ABB RAPID module: robotPath.mod

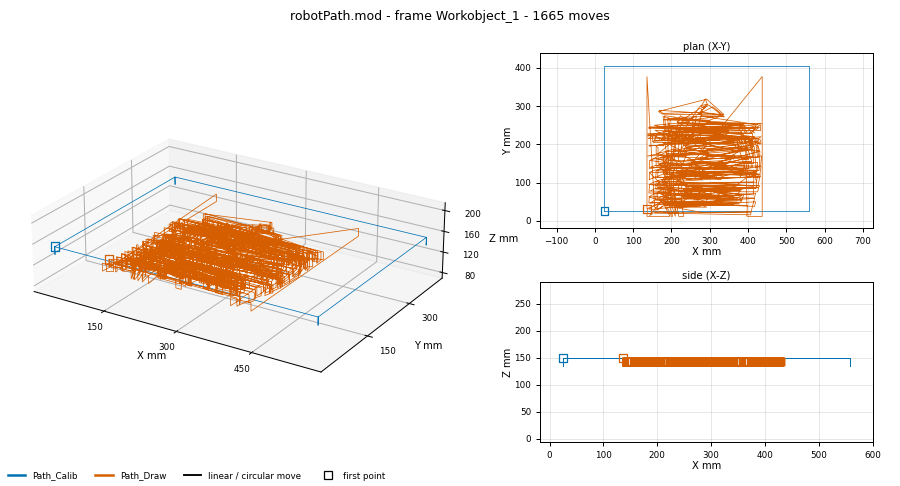
[picture p0: tool path of robotPath.mod in frame Workobject_1, 1665 of 1667 moves have a stored position in this frame; points joined in program order, loops and branches not executed]
MODULE MainModule
    CONST jointtarget home:=[[-90,40,10,0,40,90],[9E+09,9E+09,9E+09,9E+09,9E+09,9E+09]];
    CONST robtarget calib_1:=[[25,25,149.5],[0,0,1,0],[0,0,0,0],[9E+09,9E+09,9E+09,9E+09,9E+09,9E+09]];
    CONST robtarget calib_1d:=[[25,25,134.5],[0,0,1,0],[0,0,0,0],[9E+09,9E+09,9E+09,9E+09,9E+09,9E+09]];
    CONST robtarget calib_2:=[[558,25,149.5],[0,0,1,0],[0,0,0,0],[9E+09,9E+09,9E+09,9E+09,9E+09,9E+09]];
    CONST robtarget calib_2d:=[[558,25,134.5],[0,0,1,0],[0,0,0,0],[9E+09,9E+09,9E+09,9E+09,9E+09,9E+09]];
    CONST robtarget calib_3:=[[558,406,149.5],[0,0,1,0],[0,0,0,0],[9E+09,9E+09,9E+09,9E+09,9E+09,9E+09]];
    CONST robtarget calib_3d:=[[558,406,134.5],[0,0,1,0],[0,0,0,0],[9E+09,9E+09,9E+09,9E+09,9E+09,9E+09]];
    CONST robtarget calib_4:=[[25,406,149.5],[0,0,1,0],[0,0,0,0],[9E+09,9E+09,9E+09,9E+09,9E+09,9E+09]];
    CONST robtarget calib_4d:=[[25,406,134.5],[0,0,1,0],[0,0,0,0],[9E+09,9E+09,9E+09,9E+09,9E+09,9E+09]];
    CONST robtarget point_0_clearance:=[[137,31,149.5],[0,0,1,0],[0, 0, 0, 0],[9E+09,9E+09,9E+09,9E+09,9E+09,9E+09]];
    CONST robtarget point_0_contact:=[[137,31,134.5],[0,0,1,0],[0, 0, 0, 0],[9E+09,9E+09,9E+09,9E+09,9E+09,9E+09]];
    CONST robtarget point_1_contact:=[[136,12,134.5],[0,0,1,0],[0, 0, 0, 0],[9E+09,9E+09,9E+09,9E+09,9E+09,9E+09]];
    CONST robtarget point_1_clearance:=[[136,12,149.5],[0,0,1,0],[0, 0, 0, 0],[9E+09,9E+09,9E+09,9E+09,9E+09,9E+09]];
    CONST robtarget point_2_clearance:=[[196,12,149.5],[0,0,1,0],[0, 0, 0, 0],[9E+09,9E+09,9E+09,9E+09,9E+09,9E+09]];
    CONST robtarget point_2_contact:=[[196,12,134.5],[0,0,1,0],[0, 0, 0, 0],[9E+09,9E+09,9E+09,9E+09,9E+09,9E+09]];
    CONST robtarget point_3_contact:=[[185,34,134.5],[0,0,1,0],[0, 0, 0, 0],[9E+09,9E+09,9E+09,9E+09,9E+09,9E+09]];
    CONST robtarget point_3_clearance:=[[185,34,149.5],[0,0,1,0],[0, 0, 0, 0],[9E+09,9E+09,9E+09,9E+09,9E+09,9E+09]];
    CONST robtarget point_4_clearance:=[[192,30,149.5],[0,0,1,0],[0, 0, 0, 0],[9E+09,9E+09,9E+09,9E+09,9E+09,9E+09]];
    CONST robtarget point_4_contact:=[[192,30,134.5],[0,0,1,0],[0, 0, 0, 0],[9E+09,9E+09,9E+09,9E+09,9E+09,9E+09]];
    CONST robtarget point_5_contact:=[[200,12,134.5],[0,0,1,0],[0, 0, 0, 0],[9E+09,9E+09,9E+09,9E+09,9E+09,9E+09]];
    CONST robtarget point_5_clearance:=[[200,12,149.5],[0,0,1,0],[0, 0, 0, 0],[9E+09,9E+09,9E+09,9E+09,9E+09,9E+09]];
    CONST robtarget point_6_clearance:=[[203,12,149.5],[0,0,1,0],[0, 0, 0, 0],[9E+09,9E+09,9E+09,9E+09,9E+09,9E+09]];
    CONST robtarget point_6_contact:=[[203,12,134.5],[0,0,1,0],[0, 0, 0, 0],[9E+09,9E+09,9E+09,9E+09,9E+09,9E+09]];
    CONST robtarget point_7_contact:=[[195,41,134.5],[0,0,1,0],[0, 0, 0, 0],[9E+09,9E+09,9E+09,9E+09,9E+09,9E+09]];
    CONST robtarget point_7_clearance:=[[195,41,149.5],[0,0,1,0],[0, 0, 0, 0],[9E+09,9E+09,9E+09,9E+09,9E+09,9E+09]];
    CONST robtarget point_8_clearance:=[[197,51,149.5],[0,0,1,0],[0, 0, 0, 0],[9E+09,9E+09,9E+09,9E+09,9E+09,9E+09]];
    CONST robtarget point_8_contact:=[[197,51,134.5],[0,0,1,0],[0, 0, 0, 0],[9E+09,9E+09,9E+09,9E+09,9E+09,9E+09]];
    CONST robtarget point_9_contact:=[[210,12,134.5],[0,0,1,0],[0, 0, 0, 0],[9E+09,9E+09,9E+09,9E+09,9E+09,9E+09]];
    CONST robtarget point_9_clearance:=[[210,12,149.5],[0,0,1,0],[0, 0, 0, 0],[9E+09,9E+09,9E+09,9E+09,9E+09,9E+09]];
    CONST robtarget point_10_clearance:=[[206,86,149.5],[0,0,1,0],[0, 0, 0, 0],[9E+09,9E+09,9E+09,9E+09,9E+09,9E+09]];
    CONST robtarget point_10_contact:=[[206,86,134.5],[0,0,1,0],[0, 0, 0, 0],[9E+09,9E+09,9E+09,9E+09,9E+09,9E+09]];
    CONST robtarget point_11_contact:=[[219,12,134.5],[0,0,1,0],[0, 0, 0, 0],[9E+09,9E+09,9E+09,9E+09,9E+09,9E+09]];
    CONST robtarget point_11_clearance:=[[219,12,149.5],[0,0,1,0],[0, 0, 0, 0],[9E+09,9E+09,9E+09,9E+09,9E+09,9E+09]];
    CONST robtarget point_12_clearance:=[[232,12,149.5],[0,0,1,0],[0, 0, 0, 0],[9E+09,9E+09,9E+09,9E+09,9E+09,9E+09]];
    CONST robtarget point_12_contact:=[[232,12,134.5],[0,0,1,0],[0, 0, 0, 0],[9E+09,9E+09,9E+09,9E+09,9E+09,9E+09]];
    CONST robtarget point_13_contact:=[[226,51,134.5],[0,0,1,0],[0, 0, 0, 0],[9E+09,9E+09,9E+09,9E+09,9E+09,9E+09]];
    CONST robtarget point_13_clearance:=[[226,51,149.5],[0,0,1,0],[0, 0, 0, 0],[9E+09,9E+09,9E+09,9E+09,9E+09,9E+09]];
    CONST robtarget point_14_clearance:=[[398,40,149.5],[0,0,1,0],[0, 0, 0, 0],[9E+09,9E+09,9E+09,9E+09,9E+09,9E+09]];
    CONST robtarget point_14_contact:=[[398,40,134.5],[0,0,1,0],[0, 0, 0, 0],[9E+09,9E+09,9E+09,9E+09,9E+09,9E+09]];
    CONST robtarget point_15_contact:=[[397,12,134.5],[0,0,1,0],[0, 0, 0, 0],[9E+09,9E+09,9E+09,9E+09,9E+09,9E+09]];
    CONST robtarget point_15_clearance:=[[397,12,149.5],[0,0,1,0],[0, 0, 0, 0],[9E+09,9E+09,9E+09,9E+09,9E+09,9E+09]];
    CONST robtarget point_16_clearance:=[[437,12,149.5],[0,0,1,0],[0, 0, 0, 0],[9E+09,9E+09,9E+09,9E+09,9E+09,9E+09]];
    CONST robtarget point_16_contact:=[[437,12,134.5],[0,0,1,0],[0, 0, 0, 0],[9E+09,9E+09,9E+09,9E+09,9E+09,9E+09]];
    CONST robtarget point_17_contact:=[[437,377,134.5],[0,0,1,0],[0, 0, 0, 0],[9E+09,9E+09,9E+09,9E+09,9E+09,9E+09]];
    CONST robtarget point_17_clearance:=[[437,377,149.5],[0,0,1,0],[0, 0, 0, 0],[9E+09,9E+09,9E+09,9E+09,9E+09,9E+09]];
    CONST robtarget point_18_clearance:=[[143,14,149.5],[0,0,1,0],[0, 0, 0, 0],[9E+09,9E+09,9E+09,9E+09,9E+09,9E+09]];
    CONST robtarget point_18_contact:=[[143,14,134.5],[0,0,1,0],[0, 0, 0, 0],[9E+09,9E+09,9E+09,9E+09,9E+09,9E+09]];
    CONST robtarget point_19_contact:=[[153,21,134.5],[0,0,1,0],[0, 0, 0, 0],[9E+09,9E+09,9E+09,9E+09,9E+09,9E+09]];
    CONST robtarget point_19_clearance:=[[153,21,149.5],[0,0,1,0],[0, 0, 0, 0],[9E+09,9E+09,9E+09,9E+09,9E+09,9E+09]];
    CONST robtarget point_20_clearance:=[[407,16,149.5],[0,0,1,0],[0, 0, 0, 0],[9E+09,9E+09,9E+09,9E+09,9E+09,9E+09]];
    CONST robtarget point_20_contact:=[[407,16,134.5],[0,0,1,0],[0, 0, 0, 0],[9E+09,9E+09,9E+09,9E+09,9E+09,9E+09]];
    CONST robtarget point_21_contact:=[[408,23,134.5],[0,0,1,0],[0, 0, 0, 0],[9E+09,9E+09,9E+09,9E+09,9E+09,9E+09]];
    CONST robtarget point_21_clearance:=[[408,23,149.5],[0,0,1,0],[0, 0, 0, 0],[9E+09,9E+09,9E+09,9E+09,9E+09,9E+09]];
    CONST robtarget point_22_clearance:=[[157,21,149.5],[0,0,1,0],[0, 0, 0, 0],[9E+09,9E+09,9E+09,9E+09,9E+09,9E+09]];
    CONST robtarget point_22_contact:=[[157,21,134.5],[0,0,1,0],[0, 0, 0, 0],[9E+09,9E+09,9E+09,9E+09,9E+09,9E+09]];
    CONST robtarget point_23_contact:=[[157,26,134.5],[0,0,1,0],[0, 0, 0, 0],[9E+09,9E+09,9E+09,9E+09,9E+09,9E+09]];
    CONST robtarget point_23_clearance:=[[157,26,149.5],[0,0,1,0],[0, 0, 0, 0],[9E+09,9E+09,9E+09,9E+09,9E+09,9E+09]];
    CONST robtarget point_24_clearance:=[[213,21,149.5],[0,0,1,0],[0, 0, 0, 0],[9E+09,9E+09,9E+09,9E+09,9E+09,9E+09]];
    CONST robtarget point_24_contact:=[[213,21,134.5],[0,0,1,0],[0, 0, 0, 0],[9E+09,9E+09,9E+09,9E+09,9E+09,9E+09]];
    CONST robtarget point_25_contact:=[[210,35,134.5],[0,0,1,0],[0, 0, 0, 0],[9E+09,9E+09,9E+09,9E+09,9E+09,9E+09]];
    CONST robtarget point_25_clearance:=[[210,35,149.5],[0,0,1,0],[0, 0, 0, 0],[9E+09,9E+09,9E+09,9E+09,9E+09,9E+09]];
    CONST robtarget point_26_clearance:=[[281,22,149.5],[0,0,1,0],[0, 0, 0, 0],[9E+09,9E+09,9E+09,9E+09,9E+09,9E+09]];
    CONST robtarget point_26_contact:=[[281,22,134.5],[0,0,1,0],[0, 0, 0, 0],[9E+09,9E+09,9E+09,9E+09,9E+09,9E+09]];
    CONST robtarget point_27_contact:=[[292,22,134.5],[0,0,1,0],[0, 0, 0, 0],[9E+09,9E+09,9E+09,9E+09,9E+09,9E+09]];
    CONST robtarget point_27_clearance:=[[292,22,149.5],[0,0,1,0],[0, 0, 0, 0],[9E+09,9E+09,9E+09,9E+09,9E+09,9E+09]];
    CONST robtarget point_28_clearance:=[[408,24,149.5],[0,0,1,0],[0, 0, 0, 0],[9E+09,9E+09,9E+09,9E+09,9E+09,9E+09]];
    CONST robtarget point_28_contact:=[[408,24,134.5],[0,0,1,0],[0, 0, 0, 0],[9E+09,9E+09,9E+09,9E+09,9E+09,9E+09]];
    CONST robtarget point_29_contact:=[[417,59,134.5],[0,0,1,0],[0, 0, 0, 0],[9E+09,9E+09,9E+09,9E+09,9E+09,9E+09]];
    CONST robtarget point_29_clearance:=[[417,59,149.5],[0,0,1,0],[0, 0, 0, 0],[9E+09,9E+09,9E+09,9E+09,9E+09,9E+09]];
    CONST robtarget point_30_clearance:=[[156,42,149.5],[0,0,1,0],[0, 0, 0, 0],[9E+09,9E+09,9E+09,9E+09,9E+09,9E+09]];
    CONST robtarget point_30_contact:=[[156,42,134.5],[0,0,1,0],[0, 0, 0, 0],[9E+09,9E+09,9E+09,9E+09,9E+09,9E+09]];
    CONST robtarget point_31_contact:=[[141,31,134.5],[0,0,1,0],[0, 0, 0, 0],[9E+09,9E+09,9E+09,9E+09,9E+09,9E+09]];
    CONST robtarget point_31_clearance:=[[141,31,149.5],[0,0,1,0],[0, 0, 0, 0],[9E+09,9E+09,9E+09,9E+09,9E+09,9E+09]];
    CONST robtarget point_32_clearance:=[[166,30,149.5],[0,0,1,0],[0, 0, 0, 0],[9E+09,9E+09,9E+09,9E+09,9E+09,9E+09]];
    CONST robtarget point_32_contact:=[[166,30,134.5],[0,0,1,0],[0, 0, 0, 0],[9E+09,9E+09,9E+09,9E+09,9E+09,9E+09]];
    CONST robtarget point_33_contact:=[[178,39,134.5],[0,0,1,0],[0, 0, 0, 0],[9E+09,9E+09,9E+09,9E+09,9E+09,9E+09]];
    CONST robtarget point_33_clearance:=[[178,39,149.5],[0,0,1,0],[0, 0, 0, 0],[9E+09,9E+09,9E+09,9E+09,9E+09,9E+09]];
    CONST robtarget point_34_clearance:=[[164,31,149.5],[0,0,1,0],[0, 0, 0, 0],[9E+09,9E+09,9E+09,9E+09,9E+09,9E+09]];
    CONST robtarget point_34_contact:=[[164,31,134.5],[0,0,1,0],[0, 0, 0, 0],[9E+09,9E+09,9E+09,9E+09,9E+09,9E+09]];
    CONST robtarget point_35_contact:=[[156,36,134.5],[0,0,1,0],[0, 0, 0, 0],[9E+09,9E+09,9E+09,9E+09,9E+09,9E+09]];
    CONST robtarget point_35_clearance:=[[156,36,149.5],[0,0,1,0],[0, 0, 0, 0],[9E+09,9E+09,9E+09,9E+09,9E+09,9E+09]];
    CONST robtarget point_36_clearance:=[[136,377,149.5],[0,0,1,0],[0, 0, 0, 0],[9E+09,9E+09,9E+09,9E+09,9E+09,9E+09]];
    CONST robtarget point_36_contact:=[[136,377,134.5],[0,0,1,0],[0, 0, 0, 0],[9E+09,9E+09,9E+09,9E+09,9E+09,9E+09]];
    CONST robtarget point_37_contact:=[[136,32,134.5],[0,0,1,0],[0, 0, 0, 0],[9E+09,9E+09,9E+09,9E+09,9E+09,9E+09]];
    CONST robtarget point_37_clearance:=[[136,32,149.5],[0,0,1,0],[0, 0, 0, 0],[9E+09,9E+09,9E+09,9E+09,9E+09,9E+09]];
    CONST robtarget point_38_clearance:=[[164,43,149.5],[0,0,1,0],[0, 0, 0, 0],[9E+09,9E+09,9E+09,9E+09,9E+09,9E+09]];
    CONST robtarget point_38_contact:=[[164,43,134.5],[0,0,1,0],[0, 0, 0, 0],[9E+09,9E+09,9E+09,9E+09,9E+09,9E+09]];
    CONST robtarget point_39_contact:=[[164,32,134.5],[0,0,1,0],[0, 0, 0, 0],[9E+09,9E+09,9E+09,9E+09,9E+09,9E+09]];
    CONST robtarget point_39_clearance:=[[164,32,149.5],[0,0,1,0],[0, 0, 0, 0],[9E+09,9E+09,9E+09,9E+09,9E+09,9E+09]];
    CONST robtarget point_40_clearance:=[[241,40,149.5],[0,0,1,0],[0, 0, 0, 0],[9E+09,9E+09,9E+09,9E+09,9E+09,9E+09]];
    CONST robtarget point_40_contact:=[[241,40,134.5],[0,0,1,0],[0, 0, 0, 0],[9E+09,9E+09,9E+09,9E+09,9E+09,9E+09]];
    CONST robtarget point_41_contact:=[[278,39,134.5],[0,0,1,0],[0, 0, 0, 0],[9E+09,9E+09,9E+09,9E+09,9E+09,9E+09]];
    CONST robtarget point_41_clearance:=[[278,39,149.5],[0,0,1,0],[0, 0, 0, 0],[9E+09,9E+09,9E+09,9E+09,9E+09,9E+09]];
    CONST robtarget point_42_clearance:=[[185,34,149.5],[0,0,1,0],[0, 0, 0, 0],[9E+09,9E+09,9E+09,9E+09,9E+09,9E+09]];
    CONST robtarget point_42_contact:=[[185,34,134.5],[0,0,1,0],[0, 0, 0, 0],[9E+09,9E+09,9E+09,9E+09,9E+09,9E+09]];
    CONST robtarget point_43_contact:=[[180,43,134.5],[0,0,1,0],[0, 0, 0, 0],[9E+09,9E+09,9E+09,9E+09,9E+09,9E+09]];
    CONST robtarget point_43_clearance:=[[180,43,149.5],[0,0,1,0],[0, 0, 0, 0],[9E+09,9E+09,9E+09,9E+09,9E+09,9E+09]];
    CONST robtarget point_44_clearance:=[[276,42,149.5],[0,0,1,0],[0, 0, 0, 0],[9E+09,9E+09,9E+09,9E+09,9E+09,9E+09]];
    CONST robtarget point_44_contact:=[[276,42,134.5],[0,0,1,0],[0, 0, 0, 0],[9E+09,9E+09,9E+09,9E+09,9E+09,9E+09]];
    CONST robtarget point_45_contact:=[[292,36,134.5],[0,0,1,0],[0, 0, 0, 0],[9E+09,9E+09,9E+09,9E+09,9E+09,9E+09]];
    CONST robtarget point_45_clearance:=[[292,36,149.5],[0,0,1,0],[0, 0, 0, 0],[9E+09,9E+09,9E+09,9E+09,9E+09,9E+09]];
    CONST robtarget point_46_clearance:=[[196,36,149.5],[0,0,1,0],[0, 0, 0, 0],[9E+09,9E+09,9E+09,9E+09,9E+09,9E+09]];
    CONST robtarget point_46_contact:=[[196,36,134.5],[0,0,1,0],[0, 0, 0, 0],[9E+09,9E+09,9E+09,9E+09,9E+09,9E+09]];
    CONST robtarget point_47_contact:=[[192,42,134.5],[0,0,1,0],[0, 0, 0, 0],[9E+09,9E+09,9E+09,9E+09,9E+09,9E+09]];
    CONST robtarget point_47_clearance:=[[192,42,149.5],[0,0,1,0],[0, 0, 0, 0],[9E+09,9E+09,9E+09,9E+09,9E+09,9E+09]];
    CONST robtarget point_48_clearance:=[[231,41,149.5],[0,0,1,0],[0, 0, 0, 0],[9E+09,9E+09,9E+09,9E+09,9E+09,9E+09]];
    CONST robtarget point_48_contact:=[[231,41,134.5],[0,0,1,0],[0, 0, 0, 0],[9E+09,9E+09,9E+09,9E+09,9E+09,9E+09]];
    CONST robtarget point_49_contact:=[[236,38,134.5],[0,0,1,0],[0, 0, 0, 0],[9E+09,9E+09,9E+09,9E+09,9E+09,9E+09]];
    CONST robtarget point_49_clearance:=[[236,38,149.5],[0,0,1,0],[0, 0, 0, 0],[9E+09,9E+09,9E+09,9E+09,9E+09,9E+09]];
    CONST robtarget point_50_clearance:=[[239,37,149.5],[0,0,1,0],[0, 0, 0, 0],[9E+09,9E+09,9E+09,9E+09,9E+09,9E+09]];
    CONST robtarget point_50_contact:=[[239,37,134.5],[0,0,1,0],[0, 0, 0, 0],[9E+09,9E+09,9E+09,9E+09,9E+09,9E+09]];
    CONST robtarget point_51_contact:=[[234,45,134.5],[0,0,1,0],[0, 0, 0, 0],[9E+09,9E+09,9E+09,9E+09,9E+09,9E+09]];
    CONST robtarget point_51_clearance:=[[234,45,149.5],[0,0,1,0],[0, 0, 0, 0],[9E+09,9E+09,9E+09,9E+09,9E+09,9E+09]];
    CONST robtarget point_52_clearance:=[[348,42,149.5],[0,0,1,0],[0, 0, 0, 0],[9E+09,9E+09,9E+09,9E+09,9E+09,9E+09]];
    CONST robtarget point_52_contact:=[[348,42,134.5],[0,0,1,0],[0, 0, 0, 0],[9E+09,9E+09,9E+09,9E+09,9E+09,9E+09]];
    CONST robtarget point_53_contact:=[[362,42,134.5],[0,0,1,0],[0, 0, 0, 0],[9E+09,9E+09,9E+09,9E+09,9E+09,9E+09]];
    CONST robtarget point_53_clearance:=[[362,42,149.5],[0,0,1,0],[0, 0, 0, 0],[9E+09,9E+09,9E+09,9E+09,9E+09,9E+09]];
    CONST robtarget point_54_clearance:=[[239,39,149.5],[0,0,1,0],[0, 0, 0, 0],[9E+09,9E+09,9E+09,9E+09,9E+09,9E+09]];
    CONST robtarget point_54_contact:=[[239,39,134.5],[0,0,1,0],[0, 0, 0, 0],[9E+09,9E+09,9E+09,9E+09,9E+09,9E+09]];
    CONST robtarget point_55_contact:=[[244,44,134.5],[0,0,1,0],[0, 0, 0, 0],[9E+09,9E+09,9E+09,9E+09,9E+09,9E+09]];
    CONST robtarget point_55_clearance:=[[244,44,149.5],[0,0,1,0],[0, 0, 0, 0],[9E+09,9E+09,9E+09,9E+09,9E+09,9E+09]];
    CONST robtarget point_56_clearance:=[[330,44,149.5],[0,0,1,0],[0, 0, 0, 0],[9E+09,9E+09,9E+09,9E+09,9E+09,9E+09]];
    CONST robtarget point_56_contact:=[[330,44,134.5],[0,0,1,0],[0, 0, 0, 0],[9E+09,9E+09,9E+09,9E+09,9E+09,9E+09]];
    CONST robtarget point_57_contact:=[[349,46,134.5],[0,0,1,0],[0, 0, 0, 0],[9E+09,9E+09,9E+09,9E+09,9E+09,9E+09]];
    CONST robtarget point_57_clearance:=[[349,46,149.5],[0,0,1,0],[0, 0, 0, 0],[9E+09,9E+09,9E+09,9E+09,9E+09,9E+09]];
    CONST robtarget point_58_clearance:=[[420,50,149.5],[0,0,1,0],[0, 0, 0, 0],[9E+09,9E+09,9E+09,9E+09,9E+09,9E+09]];
    CONST robtarget point_58_contact:=[[420,50,134.5],[0,0,1,0],[0, 0, 0, 0],[9E+09,9E+09,9E+09,9E+09,9E+09,9E+09]];
    CONST robtarget point_59_contact:=[[417,38,134.5],[0,0,1,0],[0, 0, 0, 0],[9E+09,9E+09,9E+09,9E+09,9E+09,9E+09]];
    CONST robtarget point_59_clearance:=[[417,38,149.5],[0,0,1,0],[0, 0, 0, 0],[9E+09,9E+09,9E+09,9E+09,9E+09,9E+09]];
    CONST robtarget point_60_clearance:=[[182,48,149.5],[0,0,1,0],[0, 0, 0, 0],[9E+09,9E+09,9E+09,9E+09,9E+09,9E+09]];
    CONST robtarget point_60_contact:=[[182,48,134.5],[0,0,1,0],[0, 0, 0, 0],[9E+09,9E+09,9E+09,9E+09,9E+09,9E+09]];
    CONST robtarget point_61_contact:=[[185,39,134.5],[0,0,1,0],[0, 0, 0, 0],[9E+09,9E+09,9E+09,9E+09,9E+09,9E+09]];
    CONST robtarget point_61_clearance:=[[185,39,149.5],[0,0,1,0],[0, 0, 0, 0],[9E+09,9E+09,9E+09,9E+09,9E+09,9E+09]];
    CONST robtarget point_62_clearance:=[[287,44,149.5],[0,0,1,0],[0, 0, 0, 0],[9E+09,9E+09,9E+09,9E+09,9E+09,9E+09]];
    CONST robtarget point_62_contact:=[[287,44,134.5],[0,0,1,0],[0, 0, 0, 0],[9E+09,9E+09,9E+09,9E+09,9E+09,9E+09]];
    CONST robtarget point_63_contact:=[[295,41,134.5],[0,0,1,0],[0, 0, 0, 0],[9E+09,9E+09,9E+09,9E+09,9E+09,9E+09]];
    CONST robtarget point_63_clearance:=[[295,41,149.5],[0,0,1,0],[0, 0, 0, 0],[9E+09,9E+09,9E+09,9E+09,9E+09,9E+09]];
    CONST robtarget point_64_clearance:=[[293,41,149.5],[0,0,1,0],[0, 0, 0, 0],[9E+09,9E+09,9E+09,9E+09,9E+09,9E+09]];
    CONST robtarget point_64_contact:=[[293,41,134.5],[0,0,1,0],[0, 0, 0, 0],[9E+09,9E+09,9E+09,9E+09,9E+09,9E+09]];
    CONST robtarget point_65_contact:=[[300,42,134.5],[0,0,1,0],[0, 0, 0, 0],[9E+09,9E+09,9E+09,9E+09,9E+09,9E+09]];
    CONST robtarget point_65_clearance:=[[300,42,149.5],[0,0,1,0],[0, 0, 0, 0],[9E+09,9E+09,9E+09,9E+09,9E+09,9E+09]];
    CONST robtarget point_66_clearance:=[[396,113,149.5],[0,0,1,0],[0, 0, 0, 0],[9E+09,9E+09,9E+09,9E+09,9E+09,9E+09]];
    CONST robtarget point_66_contact:=[[396,113,134.5],[0,0,1,0],[0, 0, 0, 0],[9E+09,9E+09,9E+09,9E+09,9E+09,9E+09]];
    CONST robtarget point_67_contact:=[[397,40,134.5],[0,0,1,0],[0, 0, 0, 0],[9E+09,9E+09,9E+09,9E+09,9E+09,9E+09]];
    CONST robtarget point_67_clearance:=[[397,40,149.5],[0,0,1,0],[0, 0, 0, 0],[9E+09,9E+09,9E+09,9E+09,9E+09,9E+09]];
    CONST robtarget point_68_clearance:=[[179,41,149.5],[0,0,1,0],[0, 0, 0, 0],[9E+09,9E+09,9E+09,9E+09,9E+09,9E+09]];
    CONST robtarget point_68_contact:=[[179,41,134.5],[0,0,1,0],[0, 0, 0, 0],[9E+09,9E+09,9E+09,9E+09,9E+09,9E+09]];
    CONST robtarget point_69_contact:=[[178,51,134.5],[0,0,1,0],[0, 0, 0, 0],[9E+09,9E+09,9E+09,9E+09,9E+09,9E+09]];
    CONST robtarget point_69_clearance:=[[178,51,149.5],[0,0,1,0],[0, 0, 0, 0],[9E+09,9E+09,9E+09,9E+09,9E+09,9E+09]];
    CONST robtarget point_70_clearance:=[[347,47,149.5],[0,0,1,0],[0, 0, 0, 0],[9E+09,9E+09,9E+09,9E+09,9E+09,9E+09]];
    CONST robtarget point_70_contact:=[[347,47,134.5],[0,0,1,0],[0, 0, 0, 0],[9E+09,9E+09,9E+09,9E+09,9E+09,9E+09]];
    CONST robtarget point_71_contact:=[[374,49,134.5],[0,0,1,0],[0, 0, 0, 0],[9E+09,9E+09,9E+09,9E+09,9E+09,9E+09]];
    CONST robtarget point_71_clearance:=[[374,49,149.5],[0,0,1,0],[0, 0, 0, 0],[9E+09,9E+09,9E+09,9E+09,9E+09,9E+09]];
    CONST robtarget point_72_clearance:=[[174,52,149.5],[0,0,1,0],[0, 0, 0, 0],[9E+09,9E+09,9E+09,9E+09,9E+09,9E+09]];
    CONST robtarget point_72_contact:=[[174,52,134.5],[0,0,1,0],[0, 0, 0, 0],[9E+09,9E+09,9E+09,9E+09,9E+09,9E+09]];
    CONST robtarget point_73_contact:=[[163,44,134.5],[0,0,1,0],[0, 0, 0, 0],[9E+09,9E+09,9E+09,9E+09,9E+09,9E+09]];
    CONST robtarget point_73_clearance:=[[163,44,149.5],[0,0,1,0],[0, 0, 0, 0],[9E+09,9E+09,9E+09,9E+09,9E+09,9E+09]];
    CONST robtarget point_74_clearance:=[[232,50,149.5],[0,0,1,0],[0, 0, 0, 0],[9E+09,9E+09,9E+09,9E+09,9E+09,9E+09]];
    CONST robtarget point_74_contact:=[[232,50,134.5],[0,0,1,0],[0, 0, 0, 0],[9E+09,9E+09,9E+09,9E+09,9E+09,9E+09]];
    CONST robtarget point_75_contact:=[[246,45,134.5],[0,0,1,0],[0, 0, 0, 0],[9E+09,9E+09,9E+09,9E+09,9E+09,9E+09]];
    CONST robtarget point_75_clearance:=[[246,45,149.5],[0,0,1,0],[0, 0, 0, 0],[9E+09,9E+09,9E+09,9E+09,9E+09,9E+09]];
    CONST robtarget point_76_clearance:=[[281,44,149.5],[0,0,1,0],[0, 0, 0, 0],[9E+09,9E+09,9E+09,9E+09,9E+09,9E+09]];
    CONST robtarget point_76_contact:=[[281,44,134.5],[0,0,1,0],[0, 0, 0, 0],[9E+09,9E+09,9E+09,9E+09,9E+09,9E+09]];
    CONST robtarget point_77_contact:=[[291,47,134.5],[0,0,1,0],[0, 0, 0, 0],[9E+09,9E+09,9E+09,9E+09,9E+09,9E+09]];
    CONST robtarget point_77_clearance:=[[291,47,149.5],[0,0,1,0],[0, 0, 0, 0],[9E+09,9E+09,9E+09,9E+09,9E+09,9E+09]];
    CONST robtarget point_78_clearance:=[[321,46,149.5],[0,0,1,0],[0, 0, 0, 0],[9E+09,9E+09,9E+09,9E+09,9E+09,9E+09]];
    CONST robtarget point_78_contact:=[[321,46,134.5],[0,0,1,0],[0, 0, 0, 0],[9E+09,9E+09,9E+09,9E+09,9E+09,9E+09]];
    CONST robtarget point_79_contact:=[[330,45,134.5],[0,0,1,0],[0, 0, 0, 0],[9E+09,9E+09,9E+09,9E+09,9E+09,9E+09]];
    CONST robtarget point_79_clearance:=[[330,45,149.5],[0,0,1,0],[0, 0, 0, 0],[9E+09,9E+09,9E+09,9E+09,9E+09,9E+09]];
    CONST robtarget point_80_clearance:=[[295,45,149.5],[0,0,1,0],[0, 0, 0, 0],[9E+09,9E+09,9E+09,9E+09,9E+09,9E+09]];
    CONST robtarget point_80_contact:=[[295,45,134.5],[0,0,1,0],[0, 0, 0, 0],[9E+09,9E+09,9E+09,9E+09,9E+09,9E+09]];
    CONST robtarget point_81_contact:=[[291,51,134.5],[0,0,1,0],[0, 0, 0, 0],[9E+09,9E+09,9E+09,9E+09,9E+09,9E+09]];
    CONST robtarget point_81_clearance:=[[291,51,149.5],[0,0,1,0],[0, 0, 0, 0],[9E+09,9E+09,9E+09,9E+09,9E+09,9E+09]];
    CONST robtarget point_82_clearance:=[[327,52,149.5],[0,0,1,0],[0, 0, 0, 0],[9E+09,9E+09,9E+09,9E+09,9E+09,9E+09]];
    CONST robtarget point_82_contact:=[[327,52,134.5],[0,0,1,0],[0, 0, 0, 0],[9E+09,9E+09,9E+09,9E+09,9E+09,9E+09]];
    CONST robtarget point_83_contact:=[[332,46,134.5],[0,0,1,0],[0, 0, 0, 0],[9E+09,9E+09,9E+09,9E+09,9E+09,9E+09]];
    CONST robtarget point_83_clearance:=[[332,46,149.5],[0,0,1,0],[0, 0, 0, 0],[9E+09,9E+09,9E+09,9E+09,9E+09,9E+09]];
    CONST robtarget point_84_clearance:=[[375,45,149.5],[0,0,1,0],[0, 0, 0, 0],[9E+09,9E+09,9E+09,9E+09,9E+09,9E+09]];
    CONST robtarget point_84_contact:=[[375,45,134.5],[0,0,1,0],[0, 0, 0, 0],[9E+09,9E+09,9E+09,9E+09,9E+09,9E+09]];
    CONST robtarget point_85_contact:=[[384,53,134.5],[0,0,1,0],[0, 0, 0, 0],[9E+09,9E+09,9E+09,9E+09,9E+09,9E+09]];
    CONST robtarget point_85_clearance:=[[384,53,149.5],[0,0,1,0],[0, 0, 0, 0],[9E+09,9E+09,9E+09,9E+09,9E+09,9E+09]];
    CONST robtarget point_86_clearance:=[[144,47,149.5],[0,0,1,0],[0, 0, 0, 0],[9E+09,9E+09,9E+09,9E+09,9E+09,9E+09]];
    CONST robtarget point_86_contact:=[[144,47,134.5],[0,0,1,0],[0, 0, 0, 0],[9E+09,9E+09,9E+09,9E+09,9E+09,9E+09]];
    CONST robtarget point_87_contact:=[[158,55,134.5],[0,0,1,0],[0, 0, 0, 0],[9E+09,9E+09,9E+09,9E+09,9E+09,9E+09]];
    CONST robtarget point_87_clearance:=[[158,55,149.5],[0,0,1,0],[0, 0, 0, 0],[9E+09,9E+09,9E+09,9E+09,9E+09,9E+09]];
    CONST robtarget point_88_clearance:=[[189,52,149.5],[0,0,1,0],[0, 0, 0, 0],[9E+09,9E+09,9E+09,9E+09,9E+09,9E+09]];
    CONST robtarget point_88_contact:=[[189,52,134.5],[0,0,1,0],[0, 0, 0, 0],[9E+09,9E+09,9E+09,9E+09,9E+09,9E+09]];
    CONST robtarget point_89_contact:=[[195,48,134.5],[0,0,1,0],[0, 0, 0, 0],[9E+09,9E+09,9E+09,9E+09,9E+09,9E+09]];
    CONST robtarget point_89_clearance:=[[195,48,149.5],[0,0,1,0],[0, 0, 0, 0],[9E+09,9E+09,9E+09,9E+09,9E+09,9E+09]];
    CONST robtarget point_90_clearance:=[[142,62,149.5],[0,0,1,0],[0, 0, 0, 0],[9E+09,9E+09,9E+09,9E+09,9E+09,9E+09]];
    CONST robtarget point_90_contact:=[[142,62,134.5],[0,0,1,0],[0, 0, 0, 0],[9E+09,9E+09,9E+09,9E+09,9E+09,9E+09]];
    CONST robtarget point_91_contact:=[[141,47,134.5],[0,0,1,0],[0, 0, 0, 0],[9E+09,9E+09,9E+09,9E+09,9E+09,9E+09]];
    CONST robtarget point_91_clearance:=[[141,47,149.5],[0,0,1,0],[0, 0, 0, 0],[9E+09,9E+09,9E+09,9E+09,9E+09,9E+09]];
    CONST robtarget point_92_clearance:=[[272,52,149.5],[0,0,1,0],[0, 0, 0, 0],[9E+09,9E+09,9E+09,9E+09,9E+09,9E+09]];
    CONST robtarget point_92_contact:=[[272,52,134.5],[0,0,1,0],[0, 0, 0, 0],[9E+09,9E+09,9E+09,9E+09,9E+09,9E+09]];
    CONST robtarget point_93_contact:=[[240,51,134.5],[0,0,1,0],[0, 0, 0, 0],[9E+09,9E+09,9E+09,9E+09,9E+09,9E+09]];
    CONST robtarget point_93_clearance:=[[240,51,149.5],[0,0,1,0],[0, 0, 0, 0],[9E+09,9E+09,9E+09,9E+09,9E+09,9E+09]];
    CONST robtarget point_94_clearance:=[[202,50,149.5],[0,0,1,0],[0, 0, 0, 0],[9E+09,9E+09,9E+09,9E+09,9E+09,9E+09]];
    CONST robtarget point_94_contact:=[[202,50,134.5],[0,0,1,0],[0, 0, 0, 0],[9E+09,9E+09,9E+09,9E+09,9E+09,9E+09]];
    CONST robtarget point_95_contact:=[[199,72,134.5],[0,0,1,0],[0, 0, 0, 0],[9E+09,9E+09,9E+09,9E+09,9E+09,9E+09]];
    CONST robtarget point_95_clearance:=[[199,72,149.5],[0,0,1,0],[0, 0, 0, 0],[9E+09,9E+09,9E+09,9E+09,9E+09,9E+09]];
    CONST robtarget point_96_clearance:=[[292,51,149.5],[0,0,1,0],[0, 0, 0, 0],[9E+09,9E+09,9E+09,9E+09,9E+09,9E+09]];
    CONST robtarget point_96_contact:=[[292,51,134.5],[0,0,1,0],[0, 0, 0, 0],[9E+09,9E+09,9E+09,9E+09,9E+09,9E+09]];
    CONST robtarget point_97_contact:=[[295,68,134.5],[0,0,1,0],[0, 0, 0, 0],[9E+09,9E+09,9E+09,9E+09,9E+09,9E+09]];
    CONST robtarget point_97_clearance:=[[295,68,149.5],[0,0,1,0],[0, 0, 0, 0],[9E+09,9E+09,9E+09,9E+09,9E+09,9E+09]];
    CONST robtarget point_98_clearance:=[[331,51,149.5],[0,0,1,0],[0, 0, 0, 0],[9E+09,9E+09,9E+09,9E+09,9E+09,9E+09]];
    CONST robtarget point_98_contact:=[[331,51,134.5],[0,0,1,0],[0, 0, 0, 0],[9E+09,9E+09,9E+09,9E+09,9E+09,9E+09]];
    CONST robtarget point_99_contact:=[[326,56,134.5],[0,0,1,0],[0, 0, 0, 0],[9E+09,9E+09,9E+09,9E+09,9E+09,9E+09]];
    CONST robtarget point_99_clearance:=[[326,56,149.5],[0,0,1,0],[0, 0, 0, 0],[9E+09,9E+09,9E+09,9E+09,9E+09,9E+09]];
    CONST robtarget point_100_clearance:=[[194,115,149.5],[0,0,1,0],[0, 0, 0, 0],[9E+09,9E+09,9E+09,9E+09,9E+09,9E+09]];
    CONST robtarget point_100_contact:=[[194,115,134.5],[0,0,1,0],[0, 0, 0, 0],[9E+09,9E+09,9E+09,9E+09,9E+09,9E+09]];
    CONST robtarget point_101_contact:=[[198,52,134.5],[0,0,1,0],[0, 0, 0, 0],[9E+09,9E+09,9E+09,9E+09,9E+09,9E+09]];
    CONST robtarget point_101_clearance:=[[198,52,149.5],[0,0,1,0],[0, 0, 0, 0],[9E+09,9E+09,9E+09,9E+09,9E+09,9E+09]];
    CONST robtarget point_102_clearance:=[[226,52,149.5],[0,0,1,0],[0, 0, 0, 0],[9E+09,9E+09,9E+09,9E+09,9E+09,9E+09]];
    CONST robtarget point_102_contact:=[[226,52,134.5],[0,0,1,0],[0, 0, 0, 0],[9E+09,9E+09,9E+09,9E+09,9E+09,9E+09]];
    CONST robtarget point_103_contact:=[[228,77,134.5],[0,0,1,0],[0, 0, 0, 0],[9E+09,9E+09,9E+09,9E+09,9E+09,9E+09]];
    CONST robtarget point_103_clearance:=[[228,77,149.5],[0,0,1,0],[0, 0, 0, 0],[9E+09,9E+09,9E+09,9E+09,9E+09,9E+09]];
    CONST robtarget point_104_clearance:=[[189,53,149.5],[0,0,1,0],[0, 0, 0, 0],[9E+09,9E+09,9E+09,9E+09,9E+09,9E+09]];
    CONST robtarget point_104_contact:=[[189,53,134.5],[0,0,1,0],[0, 0, 0, 0],[9E+09,9E+09,9E+09,9E+09,9E+09,9E+09]];
    CONST robtarget point_105_contact:=[[194,60,134.5],[0,0,1,0],[0, 0, 0, 0],[9E+09,9E+09,9E+09,9E+09,9E+09,9E+09]];
    CONST robtarget point_105_clearance:=[[194,60,149.5],[0,0,1,0],[0, 0, 0, 0],[9E+09,9E+09,9E+09,9E+09,9E+09,9E+09]];
    CONST robtarget point_106_clearance:=[[235,53,149.5],[0,0,1,0],[0, 0, 0, 0],[9E+09,9E+09,9E+09,9E+09,9E+09,9E+09]];
    CONST robtarget point_106_contact:=[[235,53,134.5],[0,0,1,0],[0, 0, 0, 0],[9E+09,9E+09,9E+09,9E+09,9E+09,9E+09]];
    CONST robtarget point_107_contact:=[[235,58,134.5],[0,0,1,0],[0, 0, 0, 0],[9E+09,9E+09,9E+09,9E+09,9E+09,9E+09]];
    CONST robtarget point_107_clearance:=[[235,58,149.5],[0,0,1,0],[0, 0, 0, 0],[9E+09,9E+09,9E+09,9E+09,9E+09,9E+09]];
    CONST robtarget point_108_clearance:=[[372,55,149.5],[0,0,1,0],[0, 0, 0, 0],[9E+09,9E+09,9E+09,9E+09,9E+09,9E+09]];
    CONST robtarget point_108_contact:=[[372,55,134.5],[0,0,1,0],[0, 0, 0, 0],[9E+09,9E+09,9E+09,9E+09,9E+09,9E+09]];
    CONST robtarget point_109_contact:=[[381,59,134.5],[0,0,1,0],[0, 0, 0, 0],[9E+09,9E+09,9E+09,9E+09,9E+09,9E+09]];
    CONST robtarget point_109_clearance:=[[381,59,149.5],[0,0,1,0],[0, 0, 0, 0],[9E+09,9E+09,9E+09,9E+09,9E+09,9E+09]];
    CONST robtarget point_110_clearance:=[[382,53,149.5],[0,0,1,0],[0, 0, 0, 0],[9E+09,9E+09,9E+09,9E+09,9E+09,9E+09]];
    CONST robtarget point_110_contact:=[[382,53,134.5],[0,0,1,0],[0, 0, 0, 0],[9E+09,9E+09,9E+09,9E+09,9E+09,9E+09]];
    CONST robtarget point_111_contact:=[[389,68,134.5],[0,0,1,0],[0, 0, 0, 0],[9E+09,9E+09,9E+09,9E+09,9E+09,9E+09]];
    CONST robtarget point_111_clearance:=[[389,68,149.5],[0,0,1,0],[0, 0, 0, 0],[9E+09,9E+09,9E+09,9E+09,9E+09,9E+09]];
    CONST robtarget point_112_clearance:=[[159,55,149.5],[0,0,1,0],[0, 0, 0, 0],[9E+09,9E+09,9E+09,9E+09,9E+09,9E+09]];
    CONST robtarget point_112_contact:=[[159,55,134.5],[0,0,1,0],[0, 0, 0, 0],[9E+09,9E+09,9E+09,9E+09,9E+09,9E+09]];
    CONST robtarget point_113_contact:=[[160,72,134.5],[0,0,1,0],[0, 0, 0, 0],[9E+09,9E+09,9E+09,9E+09,9E+09,9E+09]];
    CONST robtarget point_113_clearance:=[[160,72,149.5],[0,0,1,0],[0, 0, 0, 0],[9E+09,9E+09,9E+09,9E+09,9E+09,9E+09]];
    CONST robtarget point_114_clearance:=[[202,68,149.5],[0,0,1,0],[0, 0, 0, 0],[9E+09,9E+09,9E+09,9E+09,9E+09,9E+09]];
    CONST robtarget point_114_contact:=[[202,68,134.5],[0,0,1,0],[0, 0, 0, 0],[9E+09,9E+09,9E+09,9E+09,9E+09,9E+09]];
    CONST robtarget point_115_contact:=[[204,55,134.5],[0,0,1,0],[0, 0, 0, 0],[9E+09,9E+09,9E+09,9E+09,9E+09,9E+09]];
    CONST robtarget point_115_clearance:=[[204,55,149.5],[0,0,1,0],[0, 0, 0, 0],[9E+09,9E+09,9E+09,9E+09,9E+09,9E+09]];
    CONST robtarget point_116_clearance:=[[164,75,149.5],[0,0,1,0],[0, 0, 0, 0],[9E+09,9E+09,9E+09,9E+09,9E+09,9E+09]];
    CONST robtarget point_116_contact:=[[164,75,134.5],[0,0,1,0],[0, 0, 0, 0],[9E+09,9E+09,9E+09,9E+09,9E+09,9E+09]];
    CONST robtarget point_117_contact:=[[164,56,134.5],[0,0,1,0],[0, 0, 0, 0],[9E+09,9E+09,9E+09,9E+09,9E+09,9E+09]];
    CONST robtarget point_117_clearance:=[[164,56,149.5],[0,0,1,0],[0, 0, 0, 0],[9E+09,9E+09,9E+09,9E+09,9E+09,9E+09]];
    CONST robtarget point_118_clearance:=[[373,60,149.5],[0,0,1,0],[0, 0, 0, 0],[9E+09,9E+09,9E+09,9E+09,9E+09,9E+09]];
    CONST robtarget point_118_contact:=[[373,60,134.5],[0,0,1,0],[0, 0, 0, 0],[9E+09,9E+09,9E+09,9E+09,9E+09,9E+09]];
    CONST robtarget point_119_contact:=[[342,57,134.5],[0,0,1,0],[0, 0, 0, 0],[9E+09,9E+09,9E+09,9E+09,9E+09,9E+09]];
    CONST robtarget point_119_clearance:=[[342,57,149.5],[0,0,1,0],[0, 0, 0, 0],[9E+09,9E+09,9E+09,9E+09,9E+09,9E+09]];
    CONST robtarget point_120_clearance:=[[229,64,149.5],[0,0,1,0],[0, 0, 0, 0],[9E+09,9E+09,9E+09,9E+09,9E+09,9E+09]];
    CONST robtarget point_120_contact:=[[229,64,134.5],[0,0,1,0],[0, 0, 0, 0],[9E+09,9E+09,9E+09,9E+09,9E+09,9E+09]];
    CONST robtarget point_121_contact:=[[239,57,134.5],[0,0,1,0],[0, 0, 0, 0],[9E+09,9E+09,9E+09,9E+09,9E+09,9E+09]];
    CONST robtarget point_121_clearance:=[[239,57,149.5],[0,0,1,0],[0, 0, 0, 0],[9E+09,9E+09,9E+09,9E+09,9E+09,9E+09]];
    CONST robtarget point_122_clearance:=[[242,64,149.5],[0,0,1,0],[0, 0, 0, 0],[9E+09,9E+09,9E+09,9E+09,9E+09,9E+09]];
    CONST robtarget point_122_contact:=[[242,64,134.5],[0,0,1,0],[0, 0, 0, 0],[9E+09,9E+09,9E+09,9E+09,9E+09,9E+09]];
    CONST robtarget point_123_contact:=[[260,57,134.5],[0,0,1,0],[0, 0, 0, 0],[9E+09,9E+09,9E+09,9E+09,9E+09,9E+09]];
    CONST robtarget point_123_clearance:=[[260,57,149.5],[0,0,1,0],[0, 0, 0, 0],[9E+09,9E+09,9E+09,9E+09,9E+09,9E+09]];
    CONST robtarget point_124_clearance:=[[261,58,149.5],[0,0,1,0],[0, 0, 0, 0],[9E+09,9E+09,9E+09,9E+09,9E+09,9E+09]];
    CONST robtarget point_124_contact:=[[261,58,134.5],[0,0,1,0],[0, 0, 0, 0],[9E+09,9E+09,9E+09,9E+09,9E+09,9E+09]];
    CONST robtarget point_125_contact:=[[272,59,134.5],[0,0,1,0],[0, 0, 0, 0],[9E+09,9E+09,9E+09,9E+09,9E+09,9E+09]];
    CONST robtarget point_125_clearance:=[[272,59,149.5],[0,0,1,0],[0, 0, 0, 0],[9E+09,9E+09,9E+09,9E+09,9E+09,9E+09]];
    CONST robtarget point_126_clearance:=[[317,62,149.5],[0,0,1,0],[0, 0, 0, 0],[9E+09,9E+09,9E+09,9E+09,9E+09,9E+09]];
    CONST robtarget point_126_contact:=[[317,62,134.5],[0,0,1,0],[0, 0, 0, 0],[9E+09,9E+09,9E+09,9E+09,9E+09,9E+09]];
    CONST robtarget point_127_contact:=[[327,62,134.5],[0,0,1,0],[0, 0, 0, 0],[9E+09,9E+09,9E+09,9E+09,9E+09,9E+09]];
    CONST robtarget point_127_clearance:=[[327,62,149.5],[0,0,1,0],[0, 0, 0, 0],[9E+09,9E+09,9E+09,9E+09,9E+09,9E+09]];
    CONST robtarget point_128_clearance:=[[165,59,149.5],[0,0,1,0],[0, 0, 0, 0],[9E+09,9E+09,9E+09,9E+09,9E+09,9E+09]];
    CONST robtarget point_128_contact:=[[165,59,134.5],[0,0,1,0],[0, 0, 0, 0],[9E+09,9E+09,9E+09,9E+09,9E+09,9E+09]];
    CONST robtarget point_129_contact:=[[174,64,134.5],[0,0,1,0],[0, 0, 0, 0],[9E+09,9E+09,9E+09,9E+09,9E+09,9E+09]];
    CONST robtarget point_129_clearance:=[[174,64,149.5],[0,0,1,0],[0, 0, 0, 0],[9E+09,9E+09,9E+09,9E+09,9E+09,9E+09]];
    CONST robtarget point_130_clearance:=[[189,59,149.5],[0,0,1,0],[0, 0, 0, 0],[9E+09,9E+09,9E+09,9E+09,9E+09,9E+09]];
    CONST robtarget point_130_contact:=[[189,59,134.5],[0,0,1,0],[0, 0, 0, 0],[9E+09,9E+09,9E+09,9E+09,9E+09,9E+09]];
    CONST robtarget point_131_contact:=[[185,67,134.5],[0,0,1,0],[0, 0, 0, 0],[9E+09,9E+09,9E+09,9E+09,9E+09,9E+09]];
    CONST robtarget point_131_clearance:=[[185,67,149.5],[0,0,1,0],[0, 0, 0, 0],[9E+09,9E+09,9E+09,9E+09,9E+09,9E+09]];
    CONST robtarget point_132_clearance:=[[317,63,149.5],[0,0,1,0],[0, 0, 0, 0],[9E+09,9E+09,9E+09,9E+09,9E+09,9E+09]];
    CONST robtarget point_132_contact:=[[317,63,134.5],[0,0,1,0],[0, 0, 0, 0],[9E+09,9E+09,9E+09,9E+09,9E+09,9E+09]];
    CONST robtarget point_133_contact:=[[303,61,134.5],[0,0,1,0],[0, 0, 0, 0],[9E+09,9E+09,9E+09,9E+09,9E+09,9E+09]];
    CONST robtarget point_133_clearance:=[[303,61,149.5],[0,0,1,0],[0, 0, 0, 0],[9E+09,9E+09,9E+09,9E+09,9E+09,9E+09]];
    CONST robtarget point_134_clearance:=[[416,60,149.5],[0,0,1,0],[0, 0, 0, 0],[9E+09,9E+09,9E+09,9E+09,9E+09,9E+09]];
    CONST robtarget point_134_contact:=[[416,60,134.5],[0,0,1,0],[0, 0, 0, 0],[9E+09,9E+09,9E+09,9E+09,9E+09,9E+09]];
    CONST robtarget point_135_contact:=[[420,72,134.5],[0,0,1,0],[0, 0, 0, 0],[9E+09,9E+09,9E+09,9E+09,9E+09,9E+09]];
    CONST robtarget point_135_clearance:=[[420,72,149.5],[0,0,1,0],[0, 0, 0, 0],[9E+09,9E+09,9E+09,9E+09,9E+09,9E+09]];
    CONST robtarget point_136_clearance:=[[268,61,149.5],[0,0,1,0],[0, 0, 0, 0],[9E+09,9E+09,9E+09,9E+09,9E+09,9E+09]];
    CONST robtarget point_136_contact:=[[268,61,134.5],[0,0,1,0],[0, 0, 0, 0],[9E+09,9E+09,9E+09,9E+09,9E+09,9E+09]];
    CONST robtarget point_137_contact:=[[251,63,134.5],[0,0,1,0],[0, 0, 0, 0],[9E+09,9E+09,9E+09,9E+09,9E+09,9E+09]];
    CONST robtarget point_137_clearance:=[[251,63,149.5],[0,0,1,0],[0, 0, 0, 0],[9E+09,9E+09,9E+09,9E+09,9E+09,9E+09]];
    CONST robtarget point_138_clearance:=[[383,66,149.5],[0,0,1,0],[0, 0, 0, 0],[9E+09,9E+09,9E+09,9E+09,9E+09,9E+09]];
    CONST robtarget point_138_contact:=[[383,66,134.5],[0,0,1,0],[0, 0, 0, 0],[9E+09,9E+09,9E+09,9E+09,9E+09,9E+09]];
    CONST robtarget point_139_contact:=[[372,60,134.5],[0,0,1,0],[0, 0, 0, 0],[9E+09,9E+09,9E+09,9E+09,9E+09,9E+09]];
    CONST robtarget point_139_clearance:=[[372,60,149.5],[0,0,1,0],[0, 0, 0, 0],[9E+09,9E+09,9E+09,9E+09,9E+09,9E+09]];
    CONST robtarget point_140_clearance:=[[316,75,149.5],[0,0,1,0],[0, 0, 0, 0],[9E+09,9E+09,9E+09,9E+09,9E+09,9E+09]];
    CONST robtarget point_140_contact:=[[316,75,134.5],[0,0,1,0],[0, 0, 0, 0],[9E+09,9E+09,9E+09,9E+09,9E+09,9E+09]];
    CONST robtarget point_141_contact:=[[330,64,134.5],[0,0,1,0],[0, 0, 0, 0],[9E+09,9E+09,9E+09,9E+09,9E+09,9E+09]];
    CONST robtarget point_141_clearance:=[[330,64,149.5],[0,0,1,0],[0, 0, 0, 0],[9E+09,9E+09,9E+09,9E+09,9E+09,9E+09]];
    CONST robtarget point_142_clearance:=[[343,64,149.5],[0,0,1,0],[0, 0, 0, 0],[9E+09,9E+09,9E+09,9E+09,9E+09,9E+09]];
    CONST robtarget point_142_contact:=[[343,64,134.5],[0,0,1,0],[0, 0, 0, 0],[9E+09,9E+09,9E+09,9E+09,9E+09,9E+09]];
    CONST robtarget point_143_contact:=[[355,63,134.5],[0,0,1,0],[0, 0, 0, 0],[9E+09,9E+09,9E+09,9E+09,9E+09,9E+09]];
    CONST robtarget point_143_clearance:=[[355,63,149.5],[0,0,1,0],[0, 0, 0, 0],[9E+09,9E+09,9E+09,9E+09,9E+09,9E+09]];
    CONST robtarget point_144_clearance:=[[159,73,149.5],[0,0,1,0],[0, 0, 0, 0],[9E+09,9E+09,9E+09,9E+09,9E+09,9E+09]];
    CONST robtarget point_144_contact:=[[159,73,134.5],[0,0,1,0],[0, 0, 0, 0],[9E+09,9E+09,9E+09,9E+09,9E+09,9E+09]];
    CONST robtarget point_145_contact:=[[141,63,134.5],[0,0,1,0],[0, 0, 0, 0],[9E+09,9E+09,9E+09,9E+09,9E+09,9E+09]];
    CONST robtarget point_145_clearance:=[[141,63,149.5],[0,0,1,0],[0, 0, 0, 0],[9E+09,9E+09,9E+09,9E+09,9E+09,9E+09]];
    CONST robtarget point_146_clearance:=[[193,63,149.5],[0,0,1,0],[0, 0, 0, 0],[9E+09,9E+09,9E+09,9E+09,9E+09,9E+09]];
    CONST robtarget point_146_contact:=[[193,63,134.5],[0,0,1,0],[0, 0, 0, 0],[9E+09,9E+09,9E+09,9E+09,9E+09,9E+09]];
    CONST robtarget point_147_contact:=[[190,87,134.5],[0,0,1,0],[0, 0, 0, 0],[9E+09,9E+09,9E+09,9E+09,9E+09,9E+09]];
    CONST robtarget point_147_clearance:=[[190,87,149.5],[0,0,1,0],[0, 0, 0, 0],[9E+09,9E+09,9E+09,9E+09,9E+09,9E+09]];
    CONST robtarget point_148_clearance:=[[241,73,149.5],[0,0,1,0],[0, 0, 0, 0],[9E+09,9E+09,9E+09,9E+09,9E+09,9E+09]];
    CONST robtarget point_148_contact:=[[241,73,134.5],[0,0,1,0],[0, 0, 0, 0],[9E+09,9E+09,9E+09,9E+09,9E+09,9E+09]];
    CONST robtarget point_149_contact:=[[265,64,134.5],[0,0,1,0],[0, 0, 0, 0],[9E+09,9E+09,9E+09,9E+09,9E+09,9E+09]];
    CONST robtarget point_149_clearance:=[[265,64,149.5],[0,0,1,0],[0, 0, 0, 0],[9E+09,9E+09,9E+09,9E+09,9E+09,9E+09]];
    CONST robtarget point_150_clearance:=[[306,63,149.5],[0,0,1,0],[0, 0, 0, 0],[9E+09,9E+09,9E+09,9E+09,9E+09,9E+09]];
    CONST robtarget point_150_contact:=[[306,63,134.5],[0,0,1,0],[0, 0, 0, 0],[9E+09,9E+09,9E+09,9E+09,9E+09,9E+09]];
    CONST robtarget point_151_contact:=[[304,70,134.5],[0,0,1,0],[0, 0, 0, 0],[9E+09,9E+09,9E+09,9E+09,9E+09,9E+09]];
    CONST robtarget point_151_clearance:=[[304,70,149.5],[0,0,1,0],[0, 0, 0, 0],[9E+09,9E+09,9E+09,9E+09,9E+09,9E+09]];
    CONST robtarget point_152_clearance:=[[235,74,149.5],[0,0,1,0],[0, 0, 0, 0],[9E+09,9E+09,9E+09,9E+09,9E+09,9E+09]];
    CONST robtarget point_152_contact:=[[235,74,134.5],[0,0,1,0],[0, 0, 0, 0],[9E+09,9E+09,9E+09,9E+09,9E+09,9E+09]];
    CONST robtarget point_153_contact:=[[244,64,134.5],[0,0,1,0],[0, 0, 0, 0],[9E+09,9E+09,9E+09,9E+09,9E+09,9E+09]];
    CONST robtarget point_153_clearance:=[[244,64,149.5],[0,0,1,0],[0, 0, 0, 0],[9E+09,9E+09,9E+09,9E+09,9E+09,9E+09]];
    CONST robtarget point_154_clearance:=[[264,65,149.5],[0,0,1,0],[0, 0, 0, 0],[9E+09,9E+09,9E+09,9E+09,9E+09,9E+09]];
    CONST robtarget point_154_contact:=[[264,65,134.5],[0,0,1,0],[0, 0, 0, 0],[9E+09,9E+09,9E+09,9E+09,9E+09,9E+09]];
    CONST robtarget point_155_contact:=[[279,70,134.5],[0,0,1,0],[0, 0, 0, 0],[9E+09,9E+09,9E+09,9E+09,9E+09,9E+09]];
    CONST robtarget point_155_clearance:=[[279,70,149.5],[0,0,1,0],[0, 0, 0, 0],[9E+09,9E+09,9E+09,9E+09,9E+09,9E+09]];
    CONST robtarget point_156_clearance:=[[361,65,149.5],[0,0,1,0],[0, 0, 0, 0],[9E+09,9E+09,9E+09,9E+09,9E+09,9E+09]];
    CONST robtarget point_156_contact:=[[361,65,134.5],[0,0,1,0],[0, 0, 0, 0],[9E+09,9E+09,9E+09,9E+09,9E+09,9E+09]];
    CONST robtarget point_157_contact:=[[374,70,134.5],[0,0,1,0],[0, 0, 0, 0],[9E+09,9E+09,9E+09,9E+09,9E+09,9E+09]];
    CONST robtarget point_157_clearance:=[[374,70,149.5],[0,0,1,0],[0, 0, 0, 0],[9E+09,9E+09,9E+09,9E+09,9E+09,9E+09]];
    CONST robtarget point_158_clearance:=[[218,96,149.5],[0,0,1,0],[0, 0, 0, 0],[9E+09,9E+09,9E+09,9E+09,9E+09,9E+09]];
    CONST robtarget point_158_contact:=[[218,96,134.5],[0,0,1,0],[0, 0, 0, 0],[9E+09,9E+09,9E+09,9E+09,9E+09,9E+09]];
    CONST robtarget point_159_contact:=[[219,66,134.5],[0,0,1,0],[0, 0, 0, 0],[9E+09,9E+09,9E+09,9E+09,9E+09,9E+09]];
    CONST robtarget point_159_clearance:=[[219,66,149.5],[0,0,1,0],[0, 0, 0, 0],[9E+09,9E+09,9E+09,9E+09,9E+09,9E+09]];
    CONST robtarget point_160_clearance:=[[358,66,149.5],[0,0,1,0],[0, 0, 0, 0],[9E+09,9E+09,9E+09,9E+09,9E+09,9E+09]];
    CONST robtarget point_160_contact:=[[358,66,134.5],[0,0,1,0],[0, 0, 0, 0],[9E+09,9E+09,9E+09,9E+09,9E+09,9E+09]];
    CONST robtarget point_161_contact:=[[345,67,134.5],[0,0,1,0],[0, 0, 0, 0],[9E+09,9E+09,9E+09,9E+09,9E+09,9E+09]];
    CONST robtarget point_161_clearance:=[[345,67,149.5],[0,0,1,0],[0, 0, 0, 0],[9E+09,9E+09,9E+09,9E+09,9E+09,9E+09]];
    CONST robtarget point_162_clearance:=[[177,67,149.5],[0,0,1,0],[0, 0, 0, 0],[9E+09,9E+09,9E+09,9E+09,9E+09,9E+09]];
    CONST robtarget point_162_contact:=[[177,67,134.5],[0,0,1,0],[0, 0, 0, 0],[9E+09,9E+09,9E+09,9E+09,9E+09,9E+09]];
    CONST robtarget point_163_contact:=[[180,74,134.5],[0,0,1,0],[0, 0, 0, 0],[9E+09,9E+09,9E+09,9E+09,9E+09,9E+09]];
    CONST robtarget point_163_clearance:=[[180,74,149.5],[0,0,1,0],[0, 0, 0, 0],[9E+09,9E+09,9E+09,9E+09,9E+09,9E+09]];
    CONST robtarget point_164_clearance:=[[299,68,149.5],[0,0,1,0],[0, 0, 0, 0],[9E+09,9E+09,9E+09,9E+09,9E+09,9E+09]];
    CONST robtarget point_164_contact:=[[299,68,134.5],[0,0,1,0],[0, 0, 0, 0],[9E+09,9E+09,9E+09,9E+09,9E+09,9E+09]];
    CONST robtarget point_165_contact:=[[305,77,134.5],[0,0,1,0],[0, 0, 0, 0],[9E+09,9E+09,9E+09,9E+09,9E+09,9E+09]];
    CONST robtarget point_165_clearance:=[[305,77,149.5],[0,0,1,0],[0, 0, 0, 0],[9E+09,9E+09,9E+09,9E+09,9E+09,9E+09]];
    CONST robtarget point_166_clearance:=[[345,69,149.5],[0,0,1,0],[0, 0, 0, 0],[9E+09,9E+09,9E+09,9E+09,9E+09,9E+09]];
    CONST robtarget point_166_contact:=[[345,69,134.5],[0,0,1,0],[0, 0, 0, 0],[9E+09,9E+09,9E+09,9E+09,9E+09,9E+09]];
    CONST robtarget point_167_contact:=[[368,72,134.5],[0,0,1,0],[0, 0, 0, 0],[9E+09,9E+09,9E+09,9E+09,9E+09,9E+09]];
    CONST robtarget point_167_clearance:=[[368,72,149.5],[0,0,1,0],[0, 0, 0, 0],[9E+09,9E+09,9E+09,9E+09,9E+09,9E+09]];
    CONST robtarget point_168_clearance:=[[414,68,149.5],[0,0,1,0],[0, 0, 0, 0],[9E+09,9E+09,9E+09,9E+09,9E+09,9E+09]];
    CONST robtarget point_168_contact:=[[414,68,134.5],[0,0,1,0],[0, 0, 0, 0],[9E+09,9E+09,9E+09,9E+09,9E+09,9E+09]];
    CONST robtarget point_169_contact:=[[415,88,134.5],[0,0,1,0],[0, 0, 0, 0],[9E+09,9E+09,9E+09,9E+09,9E+09,9E+09]];
    CONST robtarget point_169_clearance:=[[415,88,149.5],[0,0,1,0],[0, 0, 0, 0],[9E+09,9E+09,9E+09,9E+09,9E+09,9E+09]];
    CONST robtarget point_170_clearance:=[[292,70,149.5],[0,0,1,0],[0, 0, 0, 0],[9E+09,9E+09,9E+09,9E+09,9E+09,9E+09]];
    CONST robtarget point_170_contact:=[[292,70,134.5],[0,0,1,0],[0, 0, 0, 0],[9E+09,9E+09,9E+09,9E+09,9E+09,9E+09]];
    CONST robtarget point_171_contact:=[[285,75,134.5],[0,0,1,0],[0, 0, 0, 0],[9E+09,9E+09,9E+09,9E+09,9E+09,9E+09]];
    CONST robtarget point_171_clearance:=[[285,75,149.5],[0,0,1,0],[0, 0, 0, 0],[9E+09,9E+09,9E+09,9E+09,9E+09,9E+09]];
    CONST robtarget point_172_clearance:=[[185,81,149.5],[0,0,1,0],[0, 0, 0, 0],[9E+09,9E+09,9E+09,9E+09,9E+09,9E+09]];
    CONST robtarget point_172_contact:=[[185,81,134.5],[0,0,1,0],[0, 0, 0, 0],[9E+09,9E+09,9E+09,9E+09,9E+09,9E+09]];
    CONST robtarget point_173_contact:=[[183,71,134.5],[0,0,1,0],[0, 0, 0, 0],[9E+09,9E+09,9E+09,9E+09,9E+09,9E+09]];
    CONST robtarget point_173_clearance:=[[183,71,149.5],[0,0,1,0],[0, 0, 0, 0],[9E+09,9E+09,9E+09,9E+09,9E+09,9E+09]];
    CONST robtarget point_174_clearance:=[[271,71,149.5],[0,0,1,0],[0, 0, 0, 0],[9E+09,9E+09,9E+09,9E+09,9E+09,9E+09]];
    CONST robtarget point_174_contact:=[[271,71,134.5],[0,0,1,0],[0, 0, 0, 0],[9E+09,9E+09,9E+09,9E+09,9E+09,9E+09]];
    CONST robtarget point_175_contact:=[[272,76,134.5],[0,0,1,0],[0, 0, 0, 0],[9E+09,9E+09,9E+09,9E+09,9E+09,9E+09]];
    CONST robtarget point_175_clearance:=[[272,76,149.5],[0,0,1,0],[0, 0, 0, 0],[9E+09,9E+09,9E+09,9E+09,9E+09,9E+09]];
    CONST robtarget point_176_clearance:=[[333,77,149.5],[0,0,1,0],[0, 0, 0, 0],[9E+09,9E+09,9E+09,9E+09,9E+09,9E+09]];
    CONST robtarget point_176_contact:=[[333,77,134.5],[0,0,1,0],[0, 0, 0, 0],[9E+09,9E+09,9E+09,9E+09,9E+09,9E+09]];
    CONST robtarget point_177_contact:=[[344,71,134.5],[0,0,1,0],[0, 0, 0, 0],[9E+09,9E+09,9E+09,9E+09,9E+09,9E+09]];
    CONST robtarget point_177_clearance:=[[344,71,149.5],[0,0,1,0],[0, 0, 0, 0],[9E+09,9E+09,9E+09,9E+09,9E+09,9E+09]];
    CONST robtarget point_178_clearance:=[[374,72,149.5],[0,0,1,0],[0, 0, 0, 0],[9E+09,9E+09,9E+09,9E+09,9E+09,9E+09]];
    CONST robtarget point_178_contact:=[[374,72,134.5],[0,0,1,0],[0, 0, 0, 0],[9E+09,9E+09,9E+09,9E+09,9E+09,9E+09]];
    CONST robtarget point_179_contact:=[[380,79,134.5],[0,0,1,0],[0, 0, 0, 0],[9E+09,9E+09,9E+09,9E+09,9E+09,9E+09]];
    CONST robtarget point_179_clearance:=[[380,79,149.5],[0,0,1,0],[0, 0, 0, 0],[9E+09,9E+09,9E+09,9E+09,9E+09,9E+09]];
    CONST robtarget point_180_clearance:=[[233,78,149.5],[0,0,1,0],[0, 0, 0, 0],[9E+09,9E+09,9E+09,9E+09,9E+09,9E+09]];
    CONST robtarget point_180_contact:=[[233,78,134.5],[0,0,1,0],[0, 0, 0, 0],[9E+09,9E+09,9E+09,9E+09,9E+09,9E+09]];
    CONST robtarget point_181_contact:=[[240,73,134.5],[0,0,1,0],[0, 0, 0, 0],[9E+09,9E+09,9E+09,9E+09,9E+09,9E+09]];
    CONST robtarget point_181_clearance:=[[240,73,149.5],[0,0,1,0],[0, 0, 0, 0],[9E+09,9E+09,9E+09,9E+09,9E+09,9E+09]];
    CONST robtarget point_182_clearance:=[[274,72,149.5],[0,0,1,0],[0, 0, 0, 0],[9E+09,9E+09,9E+09,9E+09,9E+09,9E+09]];
    CONST robtarget point_182_contact:=[[274,72,134.5],[0,0,1,0],[0, 0, 0, 0],[9E+09,9E+09,9E+09,9E+09,9E+09,9E+09]];
    CONST robtarget point_183_contact:=[[275,78,134.5],[0,0,1,0],[0, 0, 0, 0],[9E+09,9E+09,9E+09,9E+09,9E+09,9E+09]];
    CONST robtarget point_183_clearance:=[[275,78,149.5],[0,0,1,0],[0, 0, 0, 0],[9E+09,9E+09,9E+09,9E+09,9E+09,9E+09]];
    CONST robtarget point_184_clearance:=[[329,76,149.5],[0,0,1,0],[0, 0, 0, 0],[9E+09,9E+09,9E+09,9E+09,9E+09,9E+09]];
    CONST robtarget point_184_contact:=[[329,76,134.5],[0,0,1,0],[0, 0, 0, 0],[9E+09,9E+09,9E+09,9E+09,9E+09,9E+09]];
    CONST robtarget point_185_contact:=[[336,73,134.5],[0,0,1,0],[0, 0, 0, 0],[9E+09,9E+09,9E+09,9E+09,9E+09,9E+09]];
    CONST robtarget point_185_clearance:=[[336,73,149.5],[0,0,1,0],[0, 0, 0, 0],[9E+09,9E+09,9E+09,9E+09,9E+09,9E+09]];
    CONST robtarget point_186_clearance:=[[143,95,149.5],[0,0,1,0],[0, 0, 0, 0],[9E+09,9E+09,9E+09,9E+09,9E+09,9E+09]];
    CONST robtarget point_186_contact:=[[143,95,134.5],[0,0,1,0],[0, 0, 0, 0],[9E+09,9E+09,9E+09,9E+09,9E+09,9E+09]];
    CONST robtarget point_187_contact:=[[141,73,134.5],[0,0,1,0],[0, 0, 0, 0],[9E+09,9E+09,9E+09,9E+09,9E+09,9E+09]];
    CONST robtarget point_187_clearance:=[[141,73,149.5],[0,0,1,0],[0, 0, 0, 0],[9E+09,9E+09,9E+09,9E+09,9E+09,9E+09]];
    CONST robtarget point_188_clearance:=[[199,73,149.5],[0,0,1,0],[0, 0, 0, 0],[9E+09,9E+09,9E+09,9E+09,9E+09,9E+09]];
    CONST robtarget point_188_contact:=[[199,73,134.5],[0,0,1,0],[0, 0, 0, 0],[9E+09,9E+09,9E+09,9E+09,9E+09,9E+09]];
    CONST robtarget point_189_contact:=[[199,127,134.5],[0,0,1,0],[0, 0, 0, 0],[9E+09,9E+09,9E+09,9E+09,9E+09,9E+09]];
    CONST robtarget point_189_clearance:=[[199,127,149.5],[0,0,1,0],[0, 0, 0, 0],[9E+09,9E+09,9E+09,9E+09,9E+09,9E+09]];
    CONST robtarget point_190_clearance:=[[251,75,149.5],[0,0,1,0],[0, 0, 0, 0],[9E+09,9E+09,9E+09,9E+09,9E+09,9E+09]];
    CONST robtarget point_190_contact:=[[251,75,134.5],[0,0,1,0],[0, 0, 0, 0],[9E+09,9E+09,9E+09,9E+09,9E+09,9E+09]];
    CONST robtarget point_191_contact:=[[256,78,134.5],[0,0,1,0],[0, 0, 0, 0],[9E+09,9E+09,9E+09,9E+09,9E+09,9E+09]];
    CONST robtarget point_191_clearance:=[[256,78,149.5],[0,0,1,0],[0, 0, 0, 0],[9E+09,9E+09,9E+09,9E+09,9E+09,9E+09]];
    CONST robtarget point_192_clearance:=[[178,83,149.5],[0,0,1,0],[0, 0, 0, 0],[9E+09,9E+09,9E+09,9E+09,9E+09,9E+09]];
    CONST robtarget point_192_contact:=[[178,83,134.5],[0,0,1,0],[0, 0, 0, 0],[9E+09,9E+09,9E+09,9E+09,9E+09,9E+09]];
    CONST robtarget point_193_contact:=[[164,75,134.5],[0,0,1,0],[0, 0, 0, 0],[9E+09,9E+09,9E+09,9E+09,9E+09,9E+09]];
    CONST robtarget point_193_clearance:=[[164,75,149.5],[0,0,1,0],[0, 0, 0, 0],[9E+09,9E+09,9E+09,9E+09,9E+09,9E+09]];
    CONST robtarget point_194_clearance:=[[180,75,149.5],[0,0,1,0],[0, 0, 0, 0],[9E+09,9E+09,9E+09,9E+09,9E+09,9E+09]];
    CONST robtarget point_194_contact:=[[180,75,134.5],[0,0,1,0],[0, 0, 0, 0],[9E+09,9E+09,9E+09,9E+09,9E+09,9E+09]];
    CONST robtarget point_195_contact:=[[180,82,134.5],[0,0,1,0],[0, 0, 0, 0],[9E+09,9E+09,9E+09,9E+09,9E+09,9E+09]];
    CONST robtarget point_195_clearance:=[[180,82,149.5],[0,0,1,0],[0, 0, 0, 0],[9E+09,9E+09,9E+09,9E+09,9E+09,9E+09]];
    CONST robtarget point_196_clearance:=[[344,75,149.5],[0,0,1,0],[0, 0, 0, 0],[9E+09,9E+09,9E+09,9E+09,9E+09,9E+09]];
    CONST robtarget point_196_contact:=[[344,75,134.5],[0,0,1,0],[0, 0, 0, 0],[9E+09,9E+09,9E+09,9E+09,9E+09,9E+09]];
    CONST robtarget point_197_contact:=[[344,81,134.5],[0,0,1,0],[0, 0, 0, 0],[9E+09,9E+09,9E+09,9E+09,9E+09,9E+09]];
    CONST robtarget point_197_clearance:=[[344,81,149.5],[0,0,1,0],[0, 0, 0, 0],[9E+09,9E+09,9E+09,9E+09,9E+09,9E+09]];
    CONST robtarget point_198_clearance:=[[252,78,149.5],[0,0,1,0],[0, 0, 0, 0],[9E+09,9E+09,9E+09,9E+09,9E+09,9E+09]];
    CONST robtarget point_198_contact:=[[252,78,134.5],[0,0,1,0],[0, 0, 0, 0],[9E+09,9E+09,9E+09,9E+09,9E+09,9E+09]];
    CONST robtarget point_199_contact:=[[242,79,134.5],[0,0,1,0],[0, 0, 0, 0],[9E+09,9E+09,9E+09,9E+09,9E+09,9E+09]];
    CONST robtarget point_199_clearance:=[[242,79,149.5],[0,0,1,0],[0, 0, 0, 0],[9E+09,9E+09,9E+09,9E+09,9E+09,9E+09]];
    CONST robtarget point_200_clearance:=[[278,78,149.5],[0,0,1,0],[0, 0, 0, 0],[9E+09,9E+09,9E+09,9E+09,9E+09,9E+09]];
    CONST robtarget point_200_contact:=[[278,78,134.5],[0,0,1,0],[0, 0, 0, 0],[9E+09,9E+09,9E+09,9E+09,9E+09,9E+09]];
    CONST robtarget point_201_contact:=[[257,79,134.5],[0,0,1,0],[0, 0, 0, 0],[9E+09,9E+09,9E+09,9E+09,9E+09,9E+09]];
    CONST robtarget point_201_clearance:=[[257,79,149.5],[0,0,1,0],[0, 0, 0, 0],[9E+09,9E+09,9E+09,9E+09,9E+09,9E+09]];
    CONST robtarget point_202_clearance:=[[278,78,149.5],[0,0,1,0],[0, 0, 0, 0],[9E+09,9E+09,9E+09,9E+09,9E+09,9E+09]];
    CONST robtarget point_202_contact:=[[278,78,134.5],[0,0,1,0],[0, 0, 0, 0],[9E+09,9E+09,9E+09,9E+09,9E+09,9E+09]];
    CONST robtarget point_203_contact:=[[284,78,134.5],[0,0,1,0],[0, 0, 0, 0],[9E+09,9E+09,9E+09,9E+09,9E+09,9E+09]];
    CONST robtarget point_203_clearance:=[[284,78,149.5],[0,0,1,0],[0, 0, 0, 0],[9E+09,9E+09,9E+09,9E+09,9E+09,9E+09]];
    CONST robtarget point_204_clearance:=[[342,76,149.5],[0,0,1,0],[0, 0, 0, 0],[9E+09,9E+09,9E+09,9E+09,9E+09,9E+09]];
    CONST robtarget point_204_contact:=[[342,76,134.5],[0,0,1,0],[0, 0, 0, 0],[9E+09,9E+09,9E+09,9E+09,9E+09,9E+09]];
    CONST robtarget point_205_contact:=[[339,81,134.5],[0,0,1,0],[0, 0, 0, 0],[9E+09,9E+09,9E+09,9E+09,9E+09,9E+09]];
    CONST robtarget point_205_clearance:=[[339,81,149.5],[0,0,1,0],[0, 0, 0, 0],[9E+09,9E+09,9E+09,9E+09,9E+09,9E+09]];
    CONST robtarget point_206_clearance:=[[428,87,149.5],[0,0,1,0],[0, 0, 0, 0],[9E+09,9E+09,9E+09,9E+09,9E+09,9E+09]];
    CONST robtarget point_206_contact:=[[428,87,134.5],[0,0,1,0],[0, 0, 0, 0],[9E+09,9E+09,9E+09,9E+09,9E+09,9E+09]];
    CONST robtarget point_207_contact:=[[425,76,134.5],[0,0,1,0],[0, 0, 0, 0],[9E+09,9E+09,9E+09,9E+09,9E+09,9E+09]];
    CONST robtarget point_207_clearance:=[[425,76,149.5],[0,0,1,0],[0, 0, 0, 0],[9E+09,9E+09,9E+09,9E+09,9E+09,9E+09]];
    CONST robtarget point_208_clearance:=[[144,78,149.5],[0,0,1,0],[0, 0, 0, 0],[9E+09,9E+09,9E+09,9E+09,9E+09,9E+09]];
    CONST robtarget point_208_contact:=[[144,78,134.5],[0,0,1,0],[0, 0, 0, 0],[9E+09,9E+09,9E+09,9E+09,9E+09,9E+09]];
    CONST robtarget point_209_contact:=[[158,85,134.5],[0,0,1,0],[0, 0, 0, 0],[9E+09,9E+09,9E+09,9E+09,9E+09,9E+09]];
    CONST robtarget point_209_clearance:=[[158,85,149.5],[0,0,1,0],[0, 0, 0, 0],[9E+09,9E+09,9E+09,9E+09,9E+09,9E+09]];
    CONST robtarget point_210_clearance:=[[228,78,149.5],[0,0,1,0],[0, 0, 0, 0],[9E+09,9E+09,9E+09,9E+09,9E+09,9E+09]];
    CONST robtarget point_210_contact:=[[228,78,134.5],[0,0,1,0],[0, 0, 0, 0],[9E+09,9E+09,9E+09,9E+09,9E+09,9E+09]];
    CONST robtarget point_211_contact:=[[222,124,134.5],[0,0,1,0],[0, 0, 0, 0],[9E+09,9E+09,9E+09,9E+09,9E+09,9E+09]];
    CONST robtarget point_211_clearance:=[[222,124,149.5],[0,0,1,0],[0, 0, 0, 0],[9E+09,9E+09,9E+09,9E+09,9E+09,9E+09]];
    CONST robtarget point_212_clearance:=[[243,81,149.5],[0,0,1,0],[0, 0, 0, 0],[9E+09,9E+09,9E+09,9E+09,9E+09,9E+09]];
    CONST robtarget point_212_contact:=[[243,81,134.5],[0,0,1,0],[0, 0, 0, 0],[9E+09,9E+09,9E+09,9E+09,9E+09,9E+09]];
    CONST robtarget point_213_contact:=[[237,80,134.5],[0,0,1,0],[0, 0, 0, 0],[9E+09,9E+09,9E+09,9E+09,9E+09,9E+09]];
    CONST robtarget point_213_clearance:=[[237,80,149.5],[0,0,1,0],[0, 0, 0, 0],[9E+09,9E+09,9E+09,9E+09,9E+09,9E+09]];
    CONST robtarget point_214_clearance:=[[342,82,149.5],[0,0,1,0],[0, 0, 0, 0],[9E+09,9E+09,9E+09,9E+09,9E+09,9E+09]];
    CONST robtarget point_214_contact:=[[342,82,134.5],[0,0,1,0],[0, 0, 0, 0],[9E+09,9E+09,9E+09,9E+09,9E+09,9E+09]];
    CONST robtarget point_215_contact:=[[331,80,134.5],[0,0,1,0],[0, 0, 0, 0],[9E+09,9E+09,9E+09,9E+09,9E+09,9E+09]];
    CONST robtarget point_215_clearance:=[[331,80,149.5],[0,0,1,0],[0, 0, 0, 0],[9E+09,9E+09,9E+09,9E+09,9E+09,9E+09]];
    CONST robtarget point_216_clearance:=[[376,79,149.5],[0,0,1,0],[0, 0, 0, 0],[9E+09,9E+09,9E+09,9E+09,9E+09,9E+09]];
    CONST robtarget point_216_contact:=[[376,79,134.5],[0,0,1,0],[0, 0, 0, 0],[9E+09,9E+09,9E+09,9E+09,9E+09,9E+09]];
    CONST robtarget point_217_contact:=[[383,82,134.5],[0,0,1,0],[0, 0, 0, 0],[9E+09,9E+09,9E+09,9E+09,9E+09,9E+09]];
    CONST robtarget point_217_clearance:=[[383,82,149.5],[0,0,1,0],[0, 0, 0, 0],[9E+09,9E+09,9E+09,9E+09,9E+09,9E+09]];
    CONST robtarget point_218_clearance:=[[238,83,149.5],[0,0,1,0],[0, 0, 0, 0],[9E+09,9E+09,9E+09,9E+09,9E+09,9E+09]];
    CONST robtarget point_218_contact:=[[238,83,134.5],[0,0,1,0],[0, 0, 0, 0],[9E+09,9E+09,9E+09,9E+09,9E+09,9E+09]];
    CONST robtarget point_219_contact:=[[231,82,134.5],[0,0,1,0],[0, 0, 0, 0],[9E+09,9E+09,9E+09,9E+09,9E+09,9E+09]];
    CONST robtarget point_219_clearance:=[[231,82,149.5],[0,0,1,0],[0, 0, 0, 0],[9E+09,9E+09,9E+09,9E+09,9E+09,9E+09]];
    CONST robtarget point_220_clearance:=[[255,79,149.5],[0,0,1,0],[0, 0, 0, 0],[9E+09,9E+09,9E+09,9E+09,9E+09,9E+09]];
    CONST robtarget point_220_contact:=[[255,79,134.5],[0,0,1,0],[0, 0, 0, 0],[9E+09,9E+09,9E+09,9E+09,9E+09,9E+09]];
    CONST robtarget point_221_contact:=[[250,86,134.5],[0,0,1,0],[0, 0, 0, 0],[9E+09,9E+09,9E+09,9E+09,9E+09,9E+09]];
    CONST robtarget point_221_clearance:=[[250,86,149.5],[0,0,1,0],[0, 0, 0, 0],[9E+09,9E+09,9E+09,9E+09,9E+09,9E+09]];
    CONST robtarget point_222_clearance:=[[348,80,149.5],[0,0,1,0],[0, 0, 0, 0],[9E+09,9E+09,9E+09,9E+09,9E+09,9E+09]];
    CONST robtarget point_222_contact:=[[348,80,134.5],[0,0,1,0],[0, 0, 0, 0],[9E+09,9E+09,9E+09,9E+09,9E+09,9E+09]];
    CONST robtarget point_223_contact:=[[353,83,134.5],[0,0,1,0],[0, 0, 0, 0],[9E+09,9E+09,9E+09,9E+09,9E+09,9E+09]];
    CONST robtarget point_223_clearance:=[[353,83,149.5],[0,0,1,0],[0, 0, 0, 0],[9E+09,9E+09,9E+09,9E+09,9E+09,9E+09]];
    CONST robtarget point_224_clearance:=[[375,81,149.5],[0,0,1,0],[0, 0, 0, 0],[9E+09,9E+09,9E+09,9E+09,9E+09,9E+09]];
    CONST robtarget point_224_contact:=[[375,81,134.5],[0,0,1,0],[0, 0, 0, 0],[9E+09,9E+09,9E+09,9E+09,9E+09,9E+09]];
    CONST robtarget point_225_contact:=[[381,84,134.5],[0,0,1,0],[0, 0, 0, 0],[9E+09,9E+09,9E+09,9E+09,9E+09,9E+09]];
    CONST robtarget point_225_clearance:=[[381,84,149.5],[0,0,1,0],[0, 0, 0, 0],[9E+09,9E+09,9E+09,9E+09,9E+09,9E+09]];
    CONST robtarget point_226_clearance:=[[364,84,149.5],[0,0,1,0],[0, 0, 0, 0],[9E+09,9E+09,9E+09,9E+09,9E+09,9E+09]];
    CONST robtarget point_226_contact:=[[364,84,134.5],[0,0,1,0],[0, 0, 0, 0],[9E+09,9E+09,9E+09,9E+09,9E+09,9E+09]];
    CONST robtarget point_227_contact:=[[353,83,134.5],[0,0,1,0],[0, 0, 0, 0],[9E+09,9E+09,9E+09,9E+09,9E+09,9E+09]];
    CONST robtarget point_227_clearance:=[[353,83,149.5],[0,0,1,0],[0, 0, 0, 0],[9E+09,9E+09,9E+09,9E+09,9E+09,9E+09]];
    CONST robtarget point_228_clearance:=[[376,83,149.5],[0,0,1,0],[0, 0, 0, 0],[9E+09,9E+09,9E+09,9E+09,9E+09,9E+09]];
    CONST robtarget point_228_contact:=[[376,83,134.5],[0,0,1,0],[0, 0, 0, 0],[9E+09,9E+09,9E+09,9E+09,9E+09,9E+09]];
    CONST robtarget point_229_contact:=[[363,87,134.5],[0,0,1,0],[0, 0, 0, 0],[9E+09,9E+09,9E+09,9E+09,9E+09,9E+09]];
    CONST robtarget point_229_clearance:=[[363,87,149.5],[0,0,1,0],[0, 0, 0, 0],[9E+09,9E+09,9E+09,9E+09,9E+09,9E+09]];
    CONST robtarget point_230_clearance:=[[240,90,149.5],[0,0,1,0],[0, 0, 0, 0],[9E+09,9E+09,9E+09,9E+09,9E+09,9E+09]];
    CONST robtarget point_230_contact:=[[240,90,134.5],[0,0,1,0],[0, 0, 0, 0],[9E+09,9E+09,9E+09,9E+09,9E+09,9E+09]];
    CONST robtarget point_231_contact:=[[249,85,134.5],[0,0,1,0],[0, 0, 0, 0],[9E+09,9E+09,9E+09,9E+09,9E+09,9E+09]];
    CONST robtarget point_231_clearance:=[[249,85,149.5],[0,0,1,0],[0, 0, 0, 0],[9E+09,9E+09,9E+09,9E+09,9E+09,9E+09]];
    CONST robtarget point_232_clearance:=[[389,85,149.5],[0,0,1,0],[0, 0, 0, 0],[9E+09,9E+09,9E+09,9E+09,9E+09,9E+09]];
    CONST robtarget point_232_contact:=[[389,85,134.5],[0,0,1,0],[0, 0, 0, 0],[9E+09,9E+09,9E+09,9E+09,9E+09,9E+09]];
    CONST robtarget point_233_contact:=[[376,87,134.5],[0,0,1,0],[0, 0, 0, 0],[9E+09,9E+09,9E+09,9E+09,9E+09,9E+09]];
    CONST robtarget point_233_clearance:=[[376,87,149.5],[0,0,1,0],[0, 0, 0, 0],[9E+09,9E+09,9E+09,9E+09,9E+09,9E+09]];
    CONST robtarget point_234_clearance:=[[159,83,149.5],[0,0,1,0],[0, 0, 0, 0],[9E+09,9E+09,9E+09,9E+09,9E+09,9E+09]];
    CONST robtarget point_234_contact:=[[159,83,134.5],[0,0,1,0],[0, 0, 0, 0],[9E+09,9E+09,9E+09,9E+09,9E+09,9E+09]];
    CONST robtarget point_235_contact:=[[160,103,134.5],[0,0,1,0],[0, 0, 0, 0],[9E+09,9E+09,9E+09,9E+09,9E+09,9E+09]];
    CONST robtarget point_235_clearance:=[[160,103,149.5],[0,0,1,0],[0, 0, 0, 0],[9E+09,9E+09,9E+09,9E+09,9E+09,9E+09]];
    CONST robtarget point_236_clearance:=[[283,85,149.5],[0,0,1,0],[0, 0, 0, 0],[9E+09,9E+09,9E+09,9E+09,9E+09,9E+09]];
    CONST robtarget point_236_contact:=[[283,85,134.5],[0,0,1,0],[0, 0, 0, 0],[9E+09,9E+09,9E+09,9E+09,9E+09,9E+09]];
    CONST robtarget point_237_contact:=[[269,91,134.5],[0,0,1,0],[0, 0, 0, 0],[9E+09,9E+09,9E+09,9E+09,9E+09,9E+09]];
    CONST robtarget point_237_clearance:=[[269,91,149.5],[0,0,1,0],[0, 0, 0, 0],[9E+09,9E+09,9E+09,9E+09,9E+09,9E+09]];
    CONST robtarget point_238_clearance:=[[421,85,149.5],[0,0,1,0],[0, 0, 0, 0],[9E+09,9E+09,9E+09,9E+09,9E+09,9E+09]];
    CONST robtarget point_238_contact:=[[421,85,134.5],[0,0,1,0],[0, 0, 0, 0],[9E+09,9E+09,9E+09,9E+09,9E+09,9E+09]];
    CONST robtarget point_239_contact:=[[423,101,134.5],[0,0,1,0],[0, 0, 0, 0],[9E+09,9E+09,9E+09,9E+09,9E+09,9E+09]];
    CONST robtarget point_239_clearance:=[[423,101,149.5],[0,0,1,0],[0, 0, 0, 0],[9E+09,9E+09,9E+09,9E+09,9E+09,9E+09]];
    CONST robtarget point_240_clearance:=[[164,96,149.5],[0,0,1,0],[0, 0, 0, 0],[9E+09,9E+09,9E+09,9E+09,9E+09,9E+09]];
    CONST robtarget point_240_contact:=[[164,96,134.5],[0,0,1,0],[0, 0, 0, 0],[9E+09,9E+09,9E+09,9E+09,9E+09,9E+09]];
    CONST robtarget point_241_contact:=[[164,86,134.5],[0,0,1,0],[0, 0, 0, 0],[9E+09,9E+09,9E+09,9E+09,9E+09,9E+09]];
    CONST robtarget point_241_clearance:=[[164,86,149.5],[0,0,1,0],[0, 0, 0, 0],[9E+09,9E+09,9E+09,9E+09,9E+09,9E+09]];
    CONST robtarget point_242_clearance:=[[190,86,149.5],[0,0,1,0],[0, 0, 0, 0],[9E+09,9E+09,9E+09,9E+09,9E+09,9E+09]];
    CONST robtarget point_242_contact:=[[190,86,134.5],[0,0,1,0],[0, 0, 0, 0],[9E+09,9E+09,9E+09,9E+09,9E+09,9E+09]];
    CONST robtarget point_243_contact:=[[187,96,134.5],[0,0,1,0],[0, 0, 0, 0],[9E+09,9E+09,9E+09,9E+09,9E+09,9E+09]];
    CONST robtarget point_243_clearance:=[[187,96,149.5],[0,0,1,0],[0, 0, 0, 0],[9E+09,9E+09,9E+09,9E+09,9E+09,9E+09]];
    CONST robtarget point_244_clearance:=[[205,130,149.5],[0,0,1,0],[0, 0, 0, 0],[9E+09,9E+09,9E+09,9E+09,9E+09,9E+09]];
    CONST robtarget point_244_contact:=[[205,130,134.5],[0,0,1,0],[0, 0, 0, 0],[9E+09,9E+09,9E+09,9E+09,9E+09,9E+09]];
    CONST robtarget point_245_contact:=[[205,86,134.5],[0,0,1,0],[0, 0, 0, 0],[9E+09,9E+09,9E+09,9E+09,9E+09,9E+09]];
    CONST robtarget point_245_clearance:=[[205,86,149.5],[0,0,1,0],[0, 0, 0, 0],[9E+09,9E+09,9E+09,9E+09,9E+09,9E+09]];
    CONST robtarget point_246_clearance:=[[165,88,149.5],[0,0,1,0],[0, 0, 0, 0],[9E+09,9E+09,9E+09,9E+09,9E+09,9E+09]];
    CONST robtarget point_246_contact:=[[165,88,134.5],[0,0,1,0],[0, 0, 0, 0],[9E+09,9E+09,9E+09,9E+09,9E+09,9E+09]];
    CONST robtarget point_247_contact:=[[178,94,134.5],[0,0,1,0],[0, 0, 0, 0],[9E+09,9E+09,9E+09,9E+09,9E+09,9E+09]];
    CONST robtarget point_247_clearance:=[[178,94,149.5],[0,0,1,0],[0, 0, 0, 0],[9E+09,9E+09,9E+09,9E+09,9E+09,9E+09]];
    CONST robtarget point_248_clearance:=[[363,89,149.5],[0,0,1,0],[0, 0, 0, 0],[9E+09,9E+09,9E+09,9E+09,9E+09,9E+09]];
    CONST robtarget point_248_contact:=[[363,89,134.5],[0,0,1,0],[0, 0, 0, 0],[9E+09,9E+09,9E+09,9E+09,9E+09,9E+09]];
    CONST robtarget point_249_contact:=[[350,87,134.5],[0,0,1,0],[0, 0, 0, 0],[9E+09,9E+09,9E+09,9E+09,9E+09,9E+09]];
    CONST robtarget point_249_clearance:=[[350,87,149.5],[0,0,1,0],[0, 0, 0, 0],[9E+09,9E+09,9E+09,9E+09,9E+09,9E+09]];
    CONST robtarget point_250_clearance:=[[427,88,149.5],[0,0,1,0],[0, 0, 0, 0],[9E+09,9E+09,9E+09,9E+09,9E+09,9E+09]];
    CONST robtarget point_250_contact:=[[427,88,134.5],[0,0,1,0],[0, 0, 0, 0],[9E+09,9E+09,9E+09,9E+09,9E+09,9E+09]];
    CONST robtarget point_251_contact:=[[431,92,134.5],[0,0,1,0],[0, 0, 0, 0],[9E+09,9E+09,9E+09,9E+09,9E+09,9E+09]];
    CONST robtarget point_251_clearance:=[[431,92,149.5],[0,0,1,0],[0, 0, 0, 0],[9E+09,9E+09,9E+09,9E+09,9E+09,9E+09]];
    CONST robtarget point_252_clearance:=[[246,93,149.5],[0,0,1,0],[0, 0, 0, 0],[9E+09,9E+09,9E+09,9E+09,9E+09,9E+09]];
    CONST robtarget point_252_contact:=[[246,93,134.5],[0,0,1,0],[0, 0, 0, 0],[9E+09,9E+09,9E+09,9E+09,9E+09,9E+09]];
    CONST robtarget point_253_contact:=[[236,89,134.5],[0,0,1,0],[0, 0, 0, 0],[9E+09,9E+09,9E+09,9E+09,9E+09,9E+09]];
    CONST robtarget point_253_clearance:=[[236,89,149.5],[0,0,1,0],[0, 0, 0, 0],[9E+09,9E+09,9E+09,9E+09,9E+09,9E+09]];
    CONST robtarget point_254_clearance:=[[268,91,149.5],[0,0,1,0],[0, 0, 0, 0],[9E+09,9E+09,9E+09,9E+09,9E+09,9E+09]];
    CONST robtarget point_254_contact:=[[268,91,134.5],[0,0,1,0],[0, 0, 0, 0],[9E+09,9E+09,9E+09,9E+09,9E+09,9E+09]];
    CONST robtarget point_255_contact:=[[247,92,134.5],[0,0,1,0],[0, 0, 0, 0],[9E+09,9E+09,9E+09,9E+09,9E+09,9E+09]];
    CONST robtarget point_255_clearance:=[[247,92,149.5],[0,0,1,0],[0, 0, 0, 0],[9E+09,9E+09,9E+09,9E+09,9E+09,9E+09]];
    CONST robtarget point_256_clearance:=[[370,94,149.5],[0,0,1,0],[0, 0, 0, 0],[9E+09,9E+09,9E+09,9E+09,9E+09,9E+09]];
    CONST robtarget point_256_contact:=[[370,94,134.5],[0,0,1,0],[0, 0, 0, 0],[9E+09,9E+09,9E+09,9E+09,9E+09,9E+09]];
    CONST robtarget point_257_contact:=[[341,93,134.5],[0,0,1,0],[0, 0, 0, 0],[9E+09,9E+09,9E+09,9E+09,9E+09,9E+09]];
    CONST robtarget point_257_clearance:=[[341,93,149.5],[0,0,1,0],[0, 0, 0, 0],[9E+09,9E+09,9E+09,9E+09,9E+09,9E+09]];
    CONST robtarget point_258_clearance:=[[370,91,149.5],[0,0,1,0],[0, 0, 0, 0],[9E+09,9E+09,9E+09,9E+09,9E+09,9E+09]];
    CONST robtarget point_258_contact:=[[370,91,134.5],[0,0,1,0],[0, 0, 0, 0],[9E+09,9E+09,9E+09,9E+09,9E+09,9E+09]];
    CONST robtarget point_259_contact:=[[375,94,134.5],[0,0,1,0],[0, 0, 0, 0],[9E+09,9E+09,9E+09,9E+09,9E+09,9E+09]];
    CONST robtarget point_259_clearance:=[[375,94,149.5],[0,0,1,0],[0, 0, 0, 0],[9E+09,9E+09,9E+09,9E+09,9E+09,9E+09]];
    CONST robtarget point_260_clearance:=[[414,90,149.5],[0,0,1,0],[0, 0, 0, 0],[9E+09,9E+09,9E+09,9E+09,9E+09,9E+09]];
    CONST robtarget point_260_contact:=[[414,90,134.5],[0,0,1,0],[0, 0, 0, 0],[9E+09,9E+09,9E+09,9E+09,9E+09,9E+09]];
    CONST robtarget point_261_contact:=[[414,101,134.5],[0,0,1,0],[0, 0, 0, 0],[9E+09,9E+09,9E+09,9E+09,9E+09,9E+09]];
    CONST robtarget point_261_clearance:=[[414,101,149.5],[0,0,1,0],[0, 0, 0, 0],[9E+09,9E+09,9E+09,9E+09,9E+09,9E+09]];
    CONST robtarget point_262_clearance:=[[180,92,149.5],[0,0,1,0],[0, 0, 0, 0],[9E+09,9E+09,9E+09,9E+09,9E+09,9E+09]];
    CONST robtarget point_262_contact:=[[180,92,134.5],[0,0,1,0],[0, 0, 0, 0],[9E+09,9E+09,9E+09,9E+09,9E+09,9E+09]];
    CONST robtarget point_263_contact:=[[178,101,134.5],[0,0,1,0],[0, 0, 0, 0],[9E+09,9E+09,9E+09,9E+09,9E+09,9E+09]];
    CONST robtarget point_263_clearance:=[[178,101,149.5],[0,0,1,0],[0, 0, 0, 0],[9E+09,9E+09,9E+09,9E+09,9E+09,9E+09]];
    CONST robtarget point_264_clearance:=[[431,117,149.5],[0,0,1,0],[0, 0, 0, 0],[9E+09,9E+09,9E+09,9E+09,9E+09,9E+09]];
    CONST robtarget point_264_contact:=[[431,117,134.5],[0,0,1,0],[0, 0, 0, 0],[9E+09,9E+09,9E+09,9E+09,9E+09,9E+09]];
    CONST robtarget point_265_contact:=[[426,92,134.5],[0,0,1,0],[0, 0, 0, 0],[9E+09,9E+09,9E+09,9E+09,9E+09,9E+09]];
    CONST robtarget point_265_clearance:=[[426,92,149.5],[0,0,1,0],[0, 0, 0, 0],[9E+09,9E+09,9E+09,9E+09,9E+09,9E+09]];
    CONST robtarget point_266_clearance:=[[160,104,149.5],[0,0,1,0],[0, 0, 0, 0],[9E+09,9E+09,9E+09,9E+09,9E+09,9E+09]];
    CONST robtarget point_266_contact:=[[160,104,134.5],[0,0,1,0],[0, 0, 0, 0],[9E+09,9E+09,9E+09,9E+09,9E+09,9E+09]];
    CONST robtarget point_267_contact:=[[141,95,134.5],[0,0,1,0],[0, 0, 0, 0],[9E+09,9E+09,9E+09,9E+09,9E+09,9E+09]];
    CONST robtarget point_267_clearance:=[[141,95,149.5],[0,0,1,0],[0, 0, 0, 0],[9E+09,9E+09,9E+09,9E+09,9E+09,9E+09]];
    CONST robtarget point_268_clearance:=[[170,97,149.5],[0,0,1,0],[0, 0, 0, 0],[9E+09,9E+09,9E+09,9E+09,9E+09,9E+09]];
    CONST robtarget point_268_contact:=[[170,97,134.5],[0,0,1,0],[0, 0, 0, 0],[9E+09,9E+09,9E+09,9E+09,9E+09,9E+09]];
    CONST robtarget point_269_contact:=[[170,94,134.5],[0,0,1,0],[0, 0, 0, 0],[9E+09,9E+09,9E+09,9E+09,9E+09,9E+09]];
    CONST robtarget point_269_clearance:=[[170,94,149.5],[0,0,1,0],[0, 0, 0, 0],[9E+09,9E+09,9E+09,9E+09,9E+09,9E+09]];
    CONST robtarget point_270_clearance:=[[167,103,149.5],[0,0,1,0],[0, 0, 0, 0],[9E+09,9E+09,9E+09,9E+09,9E+09,9E+09]];
    CONST robtarget point_270_contact:=[[167,103,134.5],[0,0,1,0],[0, 0, 0, 0],[9E+09,9E+09,9E+09,9E+09,9E+09,9E+09]];
    CONST robtarget point_271_contact:=[[164,97,134.5],[0,0,1,0],[0, 0, 0, 0],[9E+09,9E+09,9E+09,9E+09,9E+09,9E+09]];
    CONST robtarget point_271_clearance:=[[164,97,149.5],[0,0,1,0],[0, 0, 0, 0],[9E+09,9E+09,9E+09,9E+09,9E+09,9E+09]];
    CONST robtarget point_272_clearance:=[[188,96,149.5],[0,0,1,0],[0, 0, 0, 0],[9E+09,9E+09,9E+09,9E+09,9E+09,9E+09]];
    CONST robtarget point_272_contact:=[[188,96,134.5],[0,0,1,0],[0, 0, 0, 0],[9E+09,9E+09,9E+09,9E+09,9E+09,9E+09]];
    CONST robtarget point_273_contact:=[[190,151,134.5],[0,0,1,0],[0, 0, 0, 0],[9E+09,9E+09,9E+09,9E+09,9E+09,9E+09]];
    CONST robtarget point_273_clearance:=[[190,151,149.5],[0,0,1,0],[0, 0, 0, 0],[9E+09,9E+09,9E+09,9E+09,9E+09,9E+09]];
    CONST robtarget point_274_clearance:=[[182,99,149.5],[0,0,1,0],[0, 0, 0, 0],[9E+09,9E+09,9E+09,9E+09,9E+09,9E+09]];
    CONST robtarget point_274_contact:=[[182,99,134.5],[0,0,1,0],[0, 0, 0, 0],[9E+09,9E+09,9E+09,9E+09,9E+09,9E+09]];
    CONST robtarget point_275_contact:=[[174,107,134.5],[0,0,1,0],[0, 0, 0, 0],[9E+09,9E+09,9E+09,9E+09,9E+09,9E+09]];
    CONST robtarget point_275_clearance:=[[174,107,149.5],[0,0,1,0],[0, 0, 0, 0],[9E+09,9E+09,9E+09,9E+09,9E+09,9E+09]];
    CONST robtarget point_276_clearance:=[[183,106,149.5],[0,0,1,0],[0, 0, 0, 0],[9E+09,9E+09,9E+09,9E+09,9E+09,9E+09]];
    CONST robtarget point_276_contact:=[[183,106,134.5],[0,0,1,0],[0, 0, 0, 0],[9E+09,9E+09,9E+09,9E+09,9E+09,9E+09]];
    CONST robtarget point_277_contact:=[[184,98,134.5],[0,0,1,0],[0, 0, 0, 0],[9E+09,9E+09,9E+09,9E+09,9E+09,9E+09]];
    CONST robtarget point_277_clearance:=[[184,98,149.5],[0,0,1,0],[0, 0, 0, 0],[9E+09,9E+09,9E+09,9E+09,9E+09,9E+09]];
    CONST robtarget point_278_clearance:=[[415,102,149.5],[0,0,1,0],[0, 0, 0, 0],[9E+09,9E+09,9E+09,9E+09,9E+09,9E+09]];
    CONST robtarget point_278_contact:=[[415,102,134.5],[0,0,1,0],[0, 0, 0, 0],[9E+09,9E+09,9E+09,9E+09,9E+09,9E+09]];
    CONST robtarget point_279_contact:=[[415,133,134.5],[0,0,1,0],[0, 0, 0, 0],[9E+09,9E+09,9E+09,9E+09,9E+09,9E+09]];
    CONST robtarget point_279_clearance:=[[415,133,149.5],[0,0,1,0],[0, 0, 0, 0],[9E+09,9E+09,9E+09,9E+09,9E+09,9E+09]];
    CONST robtarget point_280_clearance:=[[422,102,149.5],[0,0,1,0],[0, 0, 0, 0],[9E+09,9E+09,9E+09,9E+09,9E+09,9E+09]];
    CONST robtarget point_280_contact:=[[422,102,134.5],[0,0,1,0],[0, 0, 0, 0],[9E+09,9E+09,9E+09,9E+09,9E+09,9E+09]];
    CONST robtarget point_281_contact:=[[424,114,134.5],[0,0,1,0],[0, 0, 0, 0],[9E+09,9E+09,9E+09,9E+09,9E+09,9E+09]];
    CONST robtarget point_281_clearance:=[[424,114,149.5],[0,0,1,0],[0, 0, 0, 0],[9E+09,9E+09,9E+09,9E+09,9E+09,9E+09]];
    CONST robtarget point_282_clearance:=[[172,108,149.5],[0,0,1,0],[0, 0, 0, 0],[9E+09,9E+09,9E+09,9E+09,9E+09,9E+09]];
    CONST robtarget point_282_contact:=[[172,108,134.5],[0,0,1,0],[0, 0, 0, 0],[9E+09,9E+09,9E+09,9E+09,9E+09,9E+09]];
    CONST robtarget point_283_contact:=[[164,105,134.5],[0,0,1,0],[0, 0, 0, 0],[9E+09,9E+09,9E+09,9E+09,9E+09,9E+09]];
    CONST robtarget point_283_clearance:=[[164,105,149.5],[0,0,1,0],[0, 0, 0, 0],[9E+09,9E+09,9E+09,9E+09,9E+09,9E+09]];
    CONST robtarget point_284_clearance:=[[143,126,149.5],[0,0,1,0],[0, 0, 0, 0],[9E+09,9E+09,9E+09,9E+09,9E+09,9E+09]];
    CONST robtarget point_284_contact:=[[143,126,134.5],[0,0,1,0],[0, 0, 0, 0],[9E+09,9E+09,9E+09,9E+09,9E+09,9E+09]];
    CONST robtarget point_285_contact:=[[142,107,134.5],[0,0,1,0],[0, 0, 0, 0],[9E+09,9E+09,9E+09,9E+09,9E+09,9E+09]];
    CONST robtarget point_285_clearance:=[[142,107,149.5],[0,0,1,0],[0, 0, 0, 0],[9E+09,9E+09,9E+09,9E+09,9E+09,9E+09]];
    CONST robtarget point_286_clearance:=[[144,109,149.5],[0,0,1,0],[0, 0, 0, 0],[9E+09,9E+09,9E+09,9E+09,9E+09,9E+09]];
    CONST robtarget point_286_contact:=[[144,109,134.5],[0,0,1,0],[0, 0, 0, 0],[9E+09,9E+09,9E+09,9E+09,9E+09,9E+09]];
    CONST robtarget point_287_contact:=[[158,115,134.5],[0,0,1,0],[0, 0, 0, 0],[9E+09,9E+09,9E+09,9E+09,9E+09,9E+09]];
    CONST robtarget point_287_clearance:=[[158,115,149.5],[0,0,1,0],[0, 0, 0, 0],[9E+09,9E+09,9E+09,9E+09,9E+09,9E+09]];
    CONST robtarget point_288_clearance:=[[267,110,149.5],[0,0,1,0],[0, 0, 0, 0],[9E+09,9E+09,9E+09,9E+09,9E+09,9E+09]];
    CONST robtarget point_288_contact:=[[267,110,134.5],[0,0,1,0],[0, 0, 0, 0],[9E+09,9E+09,9E+09,9E+09,9E+09,9E+09]];
    CONST robtarget point_289_contact:=[[277,109,134.5],[0,0,1,0],[0, 0, 0, 0],[9E+09,9E+09,9E+09,9E+09,9E+09,9E+09]];
    CONST robtarget point_289_clearance:=[[277,109,149.5],[0,0,1,0],[0, 0, 0, 0],[9E+09,9E+09,9E+09,9E+09,9E+09,9E+09]];
    CONST robtarget point_290_clearance:=[[280,107,149.5],[0,0,1,0],[0, 0, 0, 0],[9E+09,9E+09,9E+09,9E+09,9E+09,9E+09]];
    CONST robtarget point_290_contact:=[[280,107,134.5],[0,0,1,0],[0, 0, 0, 0],[9E+09,9E+09,9E+09,9E+09,9E+09,9E+09]];
    CONST robtarget point_291_contact:=[[276,114,134.5],[0,0,1,0],[0, 0, 0, 0],[9E+09,9E+09,9E+09,9E+09,9E+09,9E+09]];
    CONST robtarget point_291_clearance:=[[276,114,149.5],[0,0,1,0],[0, 0, 0, 0],[9E+09,9E+09,9E+09,9E+09,9E+09,9E+09]];
    CONST robtarget point_292_clearance:=[[329,108,149.5],[0,0,1,0],[0, 0, 0, 0],[9E+09,9E+09,9E+09,9E+09,9E+09,9E+09]];
    CONST robtarget point_292_contact:=[[329,108,134.5],[0,0,1,0],[0, 0, 0, 0],[9E+09,9E+09,9E+09,9E+09,9E+09,9E+09]];
    CONST robtarget point_293_contact:=[[336,115,134.5],[0,0,1,0],[0, 0, 0, 0],[9E+09,9E+09,9E+09,9E+09,9E+09,9E+09]];
    CONST robtarget point_293_clearance:=[[336,115,149.5],[0,0,1,0],[0, 0, 0, 0],[9E+09,9E+09,9E+09,9E+09,9E+09,9E+09]];
    CONST robtarget point_294_clearance:=[[240,108,149.5],[0,0,1,0],[0, 0, 0, 0],[9E+09,9E+09,9E+09,9E+09,9E+09,9E+09]];
    CONST robtarget point_294_contact:=[[240,108,134.5],[0,0,1,0],[0, 0, 0, 0],[9E+09,9E+09,9E+09,9E+09,9E+09,9E+09]];
    CONST robtarget point_295_contact:=[[235,114,134.5],[0,0,1,0],[0, 0, 0, 0],[9E+09,9E+09,9E+09,9E+09,9E+09,9E+09]];
    CONST robtarget point_295_clearance:=[[235,114,149.5],[0,0,1,0],[0, 0, 0, 0],[9E+09,9E+09,9E+09,9E+09,9E+09,9E+09]];
    CONST robtarget point_296_clearance:=[[178,110,149.5],[0,0,1,0],[0, 0, 0, 0],[9E+09,9E+09,9E+09,9E+09,9E+09,9E+09]];
    CONST robtarget point_296_contact:=[[178,110,134.5],[0,0,1,0],[0, 0, 0, 0],[9E+09,9E+09,9E+09,9E+09,9E+09,9E+09]];
    CONST robtarget point_297_contact:=[[183,115,134.5],[0,0,1,0],[0, 0, 0, 0],[9E+09,9E+09,9E+09,9E+09,9E+09,9E+09]];
    CONST robtarget point_297_clearance:=[[183,115,149.5],[0,0,1,0],[0, 0, 0, 0],[9E+09,9E+09,9E+09,9E+09,9E+09,9E+09]];
    CONST robtarget point_298_clearance:=[[250,124,149.5],[0,0,1,0],[0, 0, 0, 0],[9E+09,9E+09,9E+09,9E+09,9E+09,9E+09]];
    CONST robtarget point_298_contact:=[[250,124,134.5],[0,0,1,0],[0, 0, 0, 0],[9E+09,9E+09,9E+09,9E+09,9E+09,9E+09]];
    CONST robtarget point_299_contact:=[[264,112,134.5],[0,0,1,0],[0, 0, 0, 0],[9E+09,9E+09,9E+09,9E+09,9E+09,9E+09]];
    CONST robtarget point_299_clearance:=[[264,112,149.5],[0,0,1,0],[0, 0, 0, 0],[9E+09,9E+09,9E+09,9E+09,9E+09,9E+09]];
    CONST robtarget point_300_clearance:=[[281,112,149.5],[0,0,1,0],[0, 0, 0, 0],[9E+09,9E+09,9E+09,9E+09,9E+09,9E+09]];
    CONST robtarget point_300_contact:=[[281,112,134.5],[0,0,1,0],[0, 0, 0, 0],[9E+09,9E+09,9E+09,9E+09,9E+09,9E+09]];
    CONST robtarget point_301_contact:=[[277,126,134.5],[0,0,1,0],[0, 0, 0, 0],[9E+09,9E+09,9E+09,9E+09,9E+09,9E+09]];
    CONST robtarget point_301_clearance:=[[277,126,149.5],[0,0,1,0],[0, 0, 0, 0],[9E+09,9E+09,9E+09,9E+09,9E+09,9E+09]];
    CONST robtarget point_302_clearance:=[[290,118,149.5],[0,0,1,0],[0, 0, 0, 0],[9E+09,9E+09,9E+09,9E+09,9E+09,9E+09]];
    CONST robtarget point_302_contact:=[[290,118,134.5],[0,0,1,0],[0, 0, 0, 0],[9E+09,9E+09,9E+09,9E+09,9E+09,9E+09]];
    CONST robtarget point_303_contact:=[[313,117,134.5],[0,0,1,0],[0, 0, 0, 0],[9E+09,9E+09,9E+09,9E+09,9E+09,9E+09]];
    CONST robtarget point_303_clearance:=[[313,117,149.5],[0,0,1,0],[0, 0, 0, 0],[9E+09,9E+09,9E+09,9E+09,9E+09,9E+09]];
    CONST robtarget point_304_clearance:=[[159,113,149.5],[0,0,1,0],[0, 0, 0, 0],[9E+09,9E+09,9E+09,9E+09,9E+09,9E+09]];
    CONST robtarget point_304_contact:=[[159,113,134.5],[0,0,1,0],[0, 0, 0, 0],[9E+09,9E+09,9E+09,9E+09,9E+09,9E+09]];
    CONST robtarget point_305_contact:=[[160,132,134.5],[0,0,1,0],[0, 0, 0, 0],[9E+09,9E+09,9E+09,9E+09,9E+09,9E+09]];
    CONST robtarget point_305_clearance:=[[160,132,149.5],[0,0,1,0],[0, 0, 0, 0],[9E+09,9E+09,9E+09,9E+09,9E+09,9E+09]];
    CONST robtarget point_306_clearance:=[[268,118,149.5],[0,0,1,0],[0, 0, 0, 0],[9E+09,9E+09,9E+09,9E+09,9E+09,9E+09]];
    CONST robtarget point_306_contact:=[[268,118,134.5],[0,0,1,0],[0, 0, 0, 0],[9E+09,9E+09,9E+09,9E+09,9E+09,9E+09]];
    CONST robtarget point_307_contact:=[[275,114,134.5],[0,0,1,0],[0, 0, 0, 0],[9E+09,9E+09,9E+09,9E+09,9E+09,9E+09]];
    CONST robtarget point_307_clearance:=[[275,114,149.5],[0,0,1,0],[0, 0, 0, 0],[9E+09,9E+09,9E+09,9E+09,9E+09,9E+09]];
    CONST robtarget point_308_clearance:=[[405,113,149.5],[0,0,1,0],[0, 0, 0, 0],[9E+09,9E+09,9E+09,9E+09,9E+09,9E+09]];
    CONST robtarget point_308_contact:=[[405,113,134.5],[0,0,1,0],[0, 0, 0, 0],[9E+09,9E+09,9E+09,9E+09,9E+09,9E+09]];
    CONST robtarget point_309_contact:=[[403,122,134.5],[0,0,1,0],[0, 0, 0, 0],[9E+09,9E+09,9E+09,9E+09,9E+09,9E+09]];
    CONST robtarget point_309_clearance:=[[403,122,149.5],[0,0,1,0],[0, 0, 0, 0],[9E+09,9E+09,9E+09,9E+09,9E+09,9E+09]];
    CONST robtarget point_310_clearance:=[[427,113,149.5],[0,0,1,0],[0, 0, 0, 0],[9E+09,9E+09,9E+09,9E+09,9E+09,9E+09]];
    CONST robtarget point_310_contact:=[[427,113,134.5],[0,0,1,0],[0, 0, 0, 0],[9E+09,9E+09,9E+09,9E+09,9E+09,9E+09]];
    CONST robtarget point_311_contact:=[[426,123,134.5],[0,0,1,0],[0, 0, 0, 0],[9E+09,9E+09,9E+09,9E+09,9E+09,9E+09]];
    CONST robtarget point_311_clearance:=[[426,123,149.5],[0,0,1,0],[0, 0, 0, 0],[9E+09,9E+09,9E+09,9E+09,9E+09,9E+09]];
    CONST robtarget point_312_clearance:=[[183,115,149.5],[0,0,1,0],[0, 0, 0, 0],[9E+09,9E+09,9E+09,9E+09,9E+09,9E+09]];
    CONST robtarget point_312_contact:=[[183,115,134.5],[0,0,1,0],[0, 0, 0, 0],[9E+09,9E+09,9E+09,9E+09,9E+09,9E+09]];
    CONST robtarget point_313_contact:=[[180,122,134.5],[0,0,1,0],[0, 0, 0, 0],[9E+09,9E+09,9E+09,9E+09,9E+09,9E+09]];
    CONST robtarget point_313_clearance:=[[180,122,149.5],[0,0,1,0],[0, 0, 0, 0],[9E+09,9E+09,9E+09,9E+09,9E+09,9E+09]];
    CONST robtarget point_314_clearance:=[[229,119,149.5],[0,0,1,0],[0, 0, 0, 0],[9E+09,9E+09,9E+09,9E+09,9E+09,9E+09]];
    CONST robtarget point_314_contact:=[[229,119,134.5],[0,0,1,0],[0, 0, 0, 0],[9E+09,9E+09,9E+09,9E+09,9E+09,9E+09]];
    CONST robtarget point_315_contact:=[[234,116,134.5],[0,0,1,0],[0, 0, 0, 0],[9E+09,9E+09,9E+09,9E+09,9E+09,9E+09]];
    CONST robtarget point_315_clearance:=[[234,116,149.5],[0,0,1,0],[0, 0, 0, 0],[9E+09,9E+09,9E+09,9E+09,9E+09,9E+09]];
    CONST robtarget point_316_clearance:=[[318,115,149.5],[0,0,1,0],[0, 0, 0, 0],[9E+09,9E+09,9E+09,9E+09,9E+09,9E+09]];
    CONST robtarget point_316_contact:=[[318,115,134.5],[0,0,1,0],[0, 0, 0, 0],[9E+09,9E+09,9E+09,9E+09,9E+09,9E+09]];
    CONST robtarget point_317_contact:=[[314,121,134.5],[0,0,1,0],[0, 0, 0, 0],[9E+09,9E+09,9E+09,9E+09,9E+09,9E+09]];
    CONST robtarget point_317_clearance:=[[314,121,149.5],[0,0,1,0],[0, 0, 0, 0],[9E+09,9E+09,9E+09,9E+09,9E+09,9E+09]];
    CONST robtarget point_318_clearance:=[[335,117,149.5],[0,0,1,0],[0, 0, 0, 0],[9E+09,9E+09,9E+09,9E+09,9E+09,9E+09]];
    CONST robtarget point_318_contact:=[[335,117,134.5],[0,0,1,0],[0, 0, 0, 0],[9E+09,9E+09,9E+09,9E+09,9E+09,9E+09]];
    CONST robtarget point_319_contact:=[[347,120,134.5],[0,0,1,0],[0, 0, 0, 0],[9E+09,9E+09,9E+09,9E+09,9E+09,9E+09]];
    CONST robtarget point_319_clearance:=[[347,120,149.5],[0,0,1,0],[0, 0, 0, 0],[9E+09,9E+09,9E+09,9E+09,9E+09,9E+09]];
    CONST robtarget point_320_clearance:=[[380,125,149.5],[0,0,1,0],[0, 0, 0, 0],[9E+09,9E+09,9E+09,9E+09,9E+09,9E+09]];
    CONST robtarget point_320_contact:=[[380,125,134.5],[0,0,1,0],[0, 0, 0, 0],[9E+09,9E+09,9E+09,9E+09,9E+09,9E+09]];
    CONST robtarget point_321_contact:=[[380,115,134.5],[0,0,1,0],[0, 0, 0, 0],[9E+09,9E+09,9E+09,9E+09,9E+09,9E+09]];
    CONST robtarget point_321_clearance:=[[380,115,149.5],[0,0,1,0],[0, 0, 0, 0],[9E+09,9E+09,9E+09,9E+09,9E+09,9E+09]];
    CONST robtarget point_322_clearance:=[[391,144,149.5],[0,0,1,0],[0, 0, 0, 0],[9E+09,9E+09,9E+09,9E+09,9E+09,9E+09]];
    CONST robtarget point_322_contact:=[[391,144,134.5],[0,0,1,0],[0, 0, 0, 0],[9E+09,9E+09,9E+09,9E+09,9E+09,9E+09]];
    CONST robtarget point_323_contact:=[[396,114,134.5],[0,0,1,0],[0, 0, 0, 0],[9E+09,9E+09,9E+09,9E+09,9E+09,9E+09]];
    CONST robtarget point_323_clearance:=[[396,114,149.5],[0,0,1,0],[0, 0, 0, 0],[9E+09,9E+09,9E+09,9E+09,9E+09,9E+09]];
    CONST robtarget point_324_clearance:=[[431,122,149.5],[0,0,1,0],[0, 0, 0, 0],[9E+09,9E+09,9E+09,9E+09,9E+09,9E+09]];
    CONST robtarget point_324_contact:=[[431,122,134.5],[0,0,1,0],[0, 0, 0, 0],[9E+09,9E+09,9E+09,9E+09,9E+09,9E+09]];
    CONST robtarget point_325_contact:=[[432,115,134.5],[0,0,1,0],[0, 0, 0, 0],[9E+09,9E+09,9E+09,9E+09,9E+09,9E+09]];
    CONST robtarget point_325_clearance:=[[432,115,149.5],[0,0,1,0],[0, 0, 0, 0],[9E+09,9E+09,9E+09,9E+09,9E+09,9E+09]];
    CONST robtarget point_326_clearance:=[[165,135,149.5],[0,0,1,0],[0, 0, 0, 0],[9E+09,9E+09,9E+09,9E+09,9E+09,9E+09]];
    CONST robtarget point_326_contact:=[[165,135,134.5],[0,0,1,0],[0, 0, 0, 0],[9E+09,9E+09,9E+09,9E+09,9E+09,9E+09]];
    CONST robtarget point_327_contact:=[[164,116,134.5],[0,0,1,0],[0, 0, 0, 0],[9E+09,9E+09,9E+09,9E+09,9E+09,9E+09]];
    CONST robtarget point_327_clearance:=[[164,116,149.5],[0,0,1,0],[0, 0, 0, 0],[9E+09,9E+09,9E+09,9E+09,9E+09,9E+09]];
    CONST robtarget point_328_clearance:=[[165,117,149.5],[0,0,1,0],[0, 0, 0, 0],[9E+09,9E+09,9E+09,9E+09,9E+09,9E+09]];
    CONST robtarget point_328_contact:=[[165,117,134.5],[0,0,1,0],[0, 0, 0, 0],[9E+09,9E+09,9E+09,9E+09,9E+09,9E+09]];
    CONST robtarget point_329_contact:=[[177,122,134.5],[0,0,1,0],[0, 0, 0, 0],[9E+09,9E+09,9E+09,9E+09,9E+09,9E+09]];
    CONST robtarget point_329_clearance:=[[177,122,149.5],[0,0,1,0],[0, 0, 0, 0],[9E+09,9E+09,9E+09,9E+09,9E+09,9E+09]];
    CONST robtarget point_330_clearance:=[[197,139,149.5],[0,0,1,0],[0, 0, 0, 0],[9E+09,9E+09,9E+09,9E+09,9E+09,9E+09]];
    CONST robtarget point_330_contact:=[[197,139,134.5],[0,0,1,0],[0, 0, 0, 0],[9E+09,9E+09,9E+09,9E+09,9E+09,9E+09]];
    CONST robtarget point_331_contact:=[[194,116,134.5],[0,0,1,0],[0, 0, 0, 0],[9E+09,9E+09,9E+09,9E+09,9E+09,9E+09]];
    CONST robtarget point_331_clearance:=[[194,116,149.5],[0,0,1,0],[0, 0, 0, 0],[9E+09,9E+09,9E+09,9E+09,9E+09,9E+09]];
    CONST robtarget point_332_clearance:=[[282,128,149.5],[0,0,1,0],[0, 0, 0, 0],[9E+09,9E+09,9E+09,9E+09,9E+09,9E+09]];
    CONST robtarget point_332_contact:=[[282,128,134.5],[0,0,1,0],[0, 0, 0, 0],[9E+09,9E+09,9E+09,9E+09,9E+09,9E+09]];
    CONST robtarget point_333_contact:=[[291,120,134.5],[0,0,1,0],[0, 0, 0, 0],[9E+09,9E+09,9E+09,9E+09,9E+09,9E+09]];
    CONST robtarget point_333_clearance:=[[291,120,149.5],[0,0,1,0],[0, 0, 0, 0],[9E+09,9E+09,9E+09,9E+09,9E+09,9E+09]];
    CONST robtarget point_334_clearance:=[[226,119,149.5],[0,0,1,0],[0, 0, 0, 0],[9E+09,9E+09,9E+09,9E+09,9E+09,9E+09]];
    CONST robtarget point_334_contact:=[[226,119,134.5],[0,0,1,0],[0, 0, 0, 0],[9E+09,9E+09,9E+09,9E+09,9E+09,9E+09]];
    CONST robtarget point_335_contact:=[[225,125,134.5],[0,0,1,0],[0, 0, 0, 0],[9E+09,9E+09,9E+09,9E+09,9E+09,9E+09]];
    CONST robtarget point_335_clearance:=[[225,125,149.5],[0,0,1,0],[0, 0, 0, 0],[9E+09,9E+09,9E+09,9E+09,9E+09,9E+09]];
    CONST robtarget point_336_clearance:=[[263,122,149.5],[0,0,1,0],[0, 0, 0, 0],[9E+09,9E+09,9E+09,9E+09,9E+09,9E+09]];
    CONST robtarget point_336_contact:=[[263,122,134.5],[0,0,1,0],[0, 0, 0, 0],[9E+09,9E+09,9E+09,9E+09,9E+09,9E+09]];
    CONST robtarget point_337_contact:=[[271,119,134.5],[0,0,1,0],[0, 0, 0, 0],[9E+09,9E+09,9E+09,9E+09,9E+09,9E+09]];
    CONST robtarget point_337_clearance:=[[271,119,149.5],[0,0,1,0],[0, 0, 0, 0],[9E+09,9E+09,9E+09,9E+09,9E+09,9E+09]];
    CONST robtarget point_338_clearance:=[[309,118,149.5],[0,0,1,0],[0, 0, 0, 0],[9E+09,9E+09,9E+09,9E+09,9E+09,9E+09]];
    CONST robtarget point_338_contact:=[[309,118,134.5],[0,0,1,0],[0, 0, 0, 0],[9E+09,9E+09,9E+09,9E+09,9E+09,9E+09]];
    CONST robtarget point_339_contact:=[[309,121,134.5],[0,0,1,0],[0, 0, 0, 0],[9E+09,9E+09,9E+09,9E+09,9E+09,9E+09]];
    CONST robtarget point_339_clearance:=[[309,121,149.5],[0,0,1,0],[0, 0, 0, 0],[9E+09,9E+09,9E+09,9E+09,9E+09,9E+09]];
    CONST robtarget point_340_clearance:=[[319,120,149.5],[0,0,1,0],[0, 0, 0, 0],[9E+09,9E+09,9E+09,9E+09,9E+09,9E+09]];
    CONST robtarget point_340_contact:=[[319,120,134.5],[0,0,1,0],[0, 0, 0, 0],[9E+09,9E+09,9E+09,9E+09,9E+09,9E+09]];
    CONST robtarget point_341_contact:=[[324,129,134.5],[0,0,1,0],[0, 0, 0, 0],[9E+09,9E+09,9E+09,9E+09,9E+09,9E+09]];
    CONST robtarget point_341_clearance:=[[324,129,149.5],[0,0,1,0],[0, 0, 0, 0],[9E+09,9E+09,9E+09,9E+09,9E+09,9E+09]];
    CONST robtarget point_342_clearance:=[[233,120,149.5],[0,0,1,0],[0, 0, 0, 0],[9E+09,9E+09,9E+09,9E+09,9E+09,9E+09]];
    CONST robtarget point_342_contact:=[[233,120,134.5],[0,0,1,0],[0, 0, 0, 0],[9E+09,9E+09,9E+09,9E+09,9E+09,9E+09]];
    CONST robtarget point_343_contact:=[[232,126,134.5],[0,0,1,0],[0, 0, 0, 0],[9E+09,9E+09,9E+09,9E+09,9E+09,9E+09]];
    CONST robtarget point_343_clearance:=[[232,126,149.5],[0,0,1,0],[0, 0, 0, 0],[9E+09,9E+09,9E+09,9E+09,9E+09,9E+09]];
    CONST robtarget point_344_clearance:=[[243,124,149.5],[0,0,1,0],[0, 0, 0, 0],[9E+09,9E+09,9E+09,9E+09,9E+09,9E+09]];
    CONST robtarget point_344_contact:=[[243,124,134.5],[0,0,1,0],[0, 0, 0, 0],[9E+09,9E+09,9E+09,9E+09,9E+09,9E+09]];
    CONST robtarget point_345_contact:=[[251,120,134.5],[0,0,1,0],[0, 0, 0, 0],[9E+09,9E+09,9E+09,9E+09,9E+09,9E+09]];
    CONST robtarget point_345_clearance:=[[251,120,149.5],[0,0,1,0],[0, 0, 0, 0],[9E+09,9E+09,9E+09,9E+09,9E+09,9E+09]];
    CONST robtarget point_346_clearance:=[[296,120,149.5],[0,0,1,0],[0, 0, 0, 0],[9E+09,9E+09,9E+09,9E+09,9E+09,9E+09]];
    CONST robtarget point_346_contact:=[[296,120,134.5],[0,0,1,0],[0, 0, 0, 0],[9E+09,9E+09,9E+09,9E+09,9E+09,9E+09]];
    CONST robtarget point_347_contact:=[[296,128,134.5],[0,0,1,0],[0, 0, 0, 0],[9E+09,9E+09,9E+09,9E+09,9E+09,9E+09]];
    CONST robtarget point_347_clearance:=[[296,128,149.5],[0,0,1,0],[0, 0, 0, 0],[9E+09,9E+09,9E+09,9E+09,9E+09,9E+09]];
    CONST robtarget point_348_clearance:=[[307,123,149.5],[0,0,1,0],[0, 0, 0, 0],[9E+09,9E+09,9E+09,9E+09,9E+09,9E+09]];
    CONST robtarget point_348_contact:=[[307,123,134.5],[0,0,1,0],[0, 0, 0, 0],[9E+09,9E+09,9E+09,9E+09,9E+09,9E+09]];
    CONST robtarget point_349_contact:=[[317,127,134.5],[0,0,1,0],[0, 0, 0, 0],[9E+09,9E+09,9E+09,9E+09,9E+09,9E+09]];
    CONST robtarget point_349_clearance:=[[317,127,149.5],[0,0,1,0],[0, 0, 0, 0],[9E+09,9E+09,9E+09,9E+09,9E+09,9E+09]];
    CONST robtarget point_350_clearance:=[[434,142,149.5],[0,0,1,0],[0, 0, 0, 0],[9E+09,9E+09,9E+09,9E+09,9E+09,9E+09]];
    CONST robtarget point_350_contact:=[[434,142,134.5],[0,0,1,0],[0, 0, 0, 0],[9E+09,9E+09,9E+09,9E+09,9E+09,9E+09]];
    CONST robtarget point_351_contact:=[[431,122,134.5],[0,0,1,0],[0, 0, 0, 0],[9E+09,9E+09,9E+09,9E+09,9E+09,9E+09]];
    CONST robtarget point_351_clearance:=[[431,122,149.5],[0,0,1,0],[0, 0, 0, 0],[9E+09,9E+09,9E+09,9E+09,9E+09,9E+09]];
    CONST robtarget point_352_clearance:=[[179,123,149.5],[0,0,1,0],[0, 0, 0, 0],[9E+09,9E+09,9E+09,9E+09,9E+09,9E+09]];
    CONST robtarget point_352_contact:=[[179,123,134.5],[0,0,1,0],[0, 0, 0, 0],[9E+09,9E+09,9E+09,9E+09,9E+09,9E+09]];
    CONST robtarget point_353_contact:=[[179,133,134.5],[0,0,1,0],[0, 0, 0, 0],[9E+09,9E+09,9E+09,9E+09,9E+09,9E+09]];
    CONST robtarget point_353_clearance:=[[179,133,149.5],[0,0,1,0],[0, 0, 0, 0],[9E+09,9E+09,9E+09,9E+09,9E+09,9E+09]];
    CONST robtarget point_354_clearance:=[[422,123,149.5],[0,0,1,0],[0, 0, 0, 0],[9E+09,9E+09,9E+09,9E+09,9E+09,9E+09]];
    CONST robtarget point_354_contact:=[[422,123,134.5],[0,0,1,0],[0, 0, 0, 0],[9E+09,9E+09,9E+09,9E+09,9E+09,9E+09]];
    CONST robtarget point_355_contact:=[[421,127,134.5],[0,0,1,0],[0, 0, 0, 0],[9E+09,9E+09,9E+09,9E+09,9E+09,9E+09]];
    CONST robtarget point_355_clearance:=[[421,127,149.5],[0,0,1,0],[0, 0, 0, 0],[9E+09,9E+09,9E+09,9E+09,9E+09,9E+09]];
    CONST robtarget point_356_clearance:=[[225,124,149.5],[0,0,1,0],[0, 0, 0, 0],[9E+09,9E+09,9E+09,9E+09,9E+09,9E+09]];
    CONST robtarget point_356_contact:=[[225,124,134.5],[0,0,1,0],[0, 0, 0, 0],[9E+09,9E+09,9E+09,9E+09,9E+09,9E+09]];
    CONST robtarget point_357_contact:=[[229,140,134.5],[0,0,1,0],[0, 0, 0, 0],[9E+09,9E+09,9E+09,9E+09,9E+09,9E+09]];
    CONST robtarget point_357_clearance:=[[229,140,149.5],[0,0,1,0],[0, 0, 0, 0],[9E+09,9E+09,9E+09,9E+09,9E+09,9E+09]];
    CONST robtarget point_358_clearance:=[[157,133,149.5],[0,0,1,0],[0, 0, 0, 0],[9E+09,9E+09,9E+09,9E+09,9E+09,9E+09]];
    CONST robtarget point_358_contact:=[[157,133,134.5],[0,0,1,0],[0, 0, 0, 0],[9E+09,9E+09,9E+09,9E+09,9E+09,9E+09]];
    CONST robtarget point_359_contact:=[[142,127,134.5],[0,0,1,0],[0, 0, 0, 0],[9E+09,9E+09,9E+09,9E+09,9E+09,9E+09]];
    CONST robtarget point_359_clearance:=[[142,127,149.5],[0,0,1,0],[0, 0, 0, 0],[9E+09,9E+09,9E+09,9E+09,9E+09,9E+09]];
    CONST robtarget point_360_clearance:=[[300,127,149.5],[0,0,1,0],[0, 0, 0, 0],[9E+09,9E+09,9E+09,9E+09,9E+09,9E+09]];
    CONST robtarget point_360_contact:=[[300,127,134.5],[0,0,1,0],[0, 0, 0, 0],[9E+09,9E+09,9E+09,9E+09,9E+09,9E+09]];
    CONST robtarget point_361_contact:=[[307,126,134.5],[0,0,1,0],[0, 0, 0, 0],[9E+09,9E+09,9E+09,9E+09,9E+09,9E+09]];
    CONST robtarget point_361_clearance:=[[307,126,149.5],[0,0,1,0],[0, 0, 0, 0],[9E+09,9E+09,9E+09,9E+09,9E+09,9E+09]];
    CONST robtarget point_362_clearance:=[[184,141,149.5],[0,0,1,0],[0, 0, 0, 0],[9E+09,9E+09,9E+09,9E+09,9E+09,9E+09]];
    CONST robtarget point_362_contact:=[[184,141,134.5],[0,0,1,0],[0, 0, 0, 0],[9E+09,9E+09,9E+09,9E+09,9E+09,9E+09]];
    CONST robtarget point_363_contact:=[[184,127,134.5],[0,0,1,0],[0, 0, 0, 0],[9E+09,9E+09,9E+09,9E+09,9E+09,9E+09]];
    CONST robtarget point_363_clearance:=[[184,127,149.5],[0,0,1,0],[0, 0, 0, 0],[9E+09,9E+09,9E+09,9E+09,9E+09,9E+09]];
    CONST robtarget point_364_clearance:=[[317,130,149.5],[0,0,1,0],[0, 0, 0, 0],[9E+09,9E+09,9E+09,9E+09,9E+09,9E+09]];
    CONST robtarget point_364_contact:=[[317,130,134.5],[0,0,1,0],[0, 0, 0, 0],[9E+09,9E+09,9E+09,9E+09,9E+09,9E+09]];
    CONST robtarget point_365_contact:=[[330,128,134.5],[0,0,1,0],[0, 0, 0, 0],[9E+09,9E+09,9E+09,9E+09,9E+09,9E+09]];
    CONST robtarget point_365_clearance:=[[330,128,149.5],[0,0,1,0],[0, 0, 0, 0],[9E+09,9E+09,9E+09,9E+09,9E+09,9E+09]];
    CONST robtarget point_366_clearance:=[[343,127,149.5],[0,0,1,0],[0, 0, 0, 0],[9E+09,9E+09,9E+09,9E+09,9E+09,9E+09]];
    CONST robtarget point_366_contact:=[[343,127,134.5],[0,0,1,0],[0, 0, 0, 0],[9E+09,9E+09,9E+09,9E+09,9E+09,9E+09]];
    CONST robtarget point_367_contact:=[[356,130,134.5],[0,0,1,0],[0, 0, 0, 0],[9E+09,9E+09,9E+09,9E+09,9E+09,9E+09]];
    CONST robtarget point_367_clearance:=[[356,130,149.5],[0,0,1,0],[0, 0, 0, 0],[9E+09,9E+09,9E+09,9E+09,9E+09,9E+09]];
    CONST robtarget point_368_clearance:=[[398,127,149.5],[0,0,1,0],[0, 0, 0, 0],[9E+09,9E+09,9E+09,9E+09,9E+09,9E+09]];
    CONST robtarget point_368_contact:=[[398,127,134.5],[0,0,1,0],[0, 0, 0, 0],[9E+09,9E+09,9E+09,9E+09,9E+09,9E+09]];
    CONST robtarget point_369_contact:=[[394,165,134.5],[0,0,1,0],[0, 0, 0, 0],[9E+09,9E+09,9E+09,9E+09,9E+09,9E+09]];
    CONST robtarget point_369_clearance:=[[394,165,149.5],[0,0,1,0],[0, 0, 0, 0],[9E+09,9E+09,9E+09,9E+09,9E+09,9E+09]];
    CONST robtarget point_370_clearance:=[[275,129,149.5],[0,0,1,0],[0, 0, 0, 0],[9E+09,9E+09,9E+09,9E+09,9E+09,9E+09]];
    CONST robtarget point_370_contact:=[[275,129,134.5],[0,0,1,0],[0, 0, 0, 0],[9E+09,9E+09,9E+09,9E+09,9E+09,9E+09]];
    CONST robtarget point_371_contact:=[[257,154,134.5],[0,0,1,0],[0, 0, 0, 0],[9E+09,9E+09,9E+09,9E+09,9E+09,9E+09]];
    CONST robtarget point_371_clearance:=[[257,154,149.5],[0,0,1,0],[0, 0, 0, 0],[9E+09,9E+09,9E+09,9E+09,9E+09,9E+09]];
    CONST robtarget point_372_clearance:=[[282,134,149.5],[0,0,1,0],[0, 0, 0, 0],[9E+09,9E+09,9E+09,9E+09,9E+09,9E+09]];
    CONST robtarget point_372_contact:=[[282,134,134.5],[0,0,1,0],[0, 0, 0, 0],[9E+09,9E+09,9E+09,9E+09,9E+09,9E+09]];
    CONST robtarget point_373_contact:=[[280,128,134.5],[0,0,1,0],[0, 0, 0, 0],[9E+09,9E+09,9E+09,9E+09,9E+09,9E+09]];
    CONST robtarget point_373_clearance:=[[280,128,149.5],[0,0,1,0],[0, 0, 0, 0],[9E+09,9E+09,9E+09,9E+09,9E+09,9E+09]];
    CONST robtarget point_374_clearance:=[[386,130,149.5],[0,0,1,0],[0, 0, 0, 0],[9E+09,9E+09,9E+09,9E+09,9E+09,9E+09]];
    CONST robtarget point_374_contact:=[[386,130,134.5],[0,0,1,0],[0, 0, 0, 0],[9E+09,9E+09,9E+09,9E+09,9E+09,9E+09]];
    CONST robtarget point_375_contact:=[[391,128,134.5],[0,0,1,0],[0, 0, 0, 0],[9E+09,9E+09,9E+09,9E+09,9E+09,9E+09]];
    CONST robtarget point_375_clearance:=[[391,128,149.5],[0,0,1,0],[0, 0, 0, 0],[9E+09,9E+09,9E+09,9E+09,9E+09,9E+09]];
    CONST robtarget point_376_clearance:=[[422,128,149.5],[0,0,1,0],[0, 0, 0, 0],[9E+09,9E+09,9E+09,9E+09,9E+09,9E+09]];
    CONST robtarget point_376_contact:=[[422,128,134.5],[0,0,1,0],[0, 0, 0, 0],[9E+09,9E+09,9E+09,9E+09,9E+09,9E+09]];
    CONST robtarget point_377_contact:=[[416,195,134.5],[0,0,1,0],[0, 0, 0, 0],[9E+09,9E+09,9E+09,9E+09,9E+09,9E+09]];
    CONST robtarget point_377_clearance:=[[416,195,149.5],[0,0,1,0],[0, 0, 0, 0],[9E+09,9E+09,9E+09,9E+09,9E+09,9E+09]];
    CONST robtarget point_378_clearance:=[[178,131,149.5],[0,0,1,0],[0, 0, 0, 0],[9E+09,9E+09,9E+09,9E+09,9E+09,9E+09]];
    CONST robtarget point_378_contact:=[[178,131,134.5],[0,0,1,0],[0, 0, 0, 0],[9E+09,9E+09,9E+09,9E+09,9E+09,9E+09]];
    CONST robtarget point_379_contact:=[[173,135,134.5],[0,0,1,0],[0, 0, 0, 0],[9E+09,9E+09,9E+09,9E+09,9E+09,9E+09]];
    CONST robtarget point_379_clearance:=[[173,135,149.5],[0,0,1,0],[0, 0, 0, 0],[9E+09,9E+09,9E+09,9E+09,9E+09,9E+09]];
    CONST robtarget point_380_clearance:=[[208,137,149.5],[0,0,1,0],[0, 0, 0, 0],[9E+09,9E+09,9E+09,9E+09,9E+09,9E+09]];
    CONST robtarget point_380_contact:=[[208,137,134.5],[0,0,1,0],[0, 0, 0, 0],[9E+09,9E+09,9E+09,9E+09,9E+09,9E+09]];
    CONST robtarget point_381_contact:=[[205,129,134.5],[0,0,1,0],[0, 0, 0, 0],[9E+09,9E+09,9E+09,9E+09,9E+09,9E+09]];
    CONST robtarget point_381_clearance:=[[205,129,149.5],[0,0,1,0],[0, 0, 0, 0],[9E+09,9E+09,9E+09,9E+09,9E+09,9E+09]];
    CONST robtarget point_382_clearance:=[[212,152,149.5],[0,0,1,0],[0, 0, 0, 0],[9E+09,9E+09,9E+09,9E+09,9E+09,9E+09]];
    CONST robtarget point_382_contact:=[[212,152,134.5],[0,0,1,0],[0, 0, 0, 0],[9E+09,9E+09,9E+09,9E+09,9E+09,9E+09]];
    CONST robtarget point_383_contact:=[[213,130,134.5],[0,0,1,0],[0, 0, 0, 0],[9E+09,9E+09,9E+09,9E+09,9E+09,9E+09]];
    CONST robtarget point_383_clearance:=[[213,130,149.5],[0,0,1,0],[0, 0, 0, 0],[9E+09,9E+09,9E+09,9E+09,9E+09,9E+09]];
    CONST robtarget point_384_clearance:=[[303,137,149.5],[0,0,1,0],[0, 0, 0, 0],[9E+09,9E+09,9E+09,9E+09,9E+09,9E+09]];
    CONST robtarget point_384_contact:=[[303,137,134.5],[0,0,1,0],[0, 0, 0, 0],[9E+09,9E+09,9E+09,9E+09,9E+09,9E+09]];
    CONST robtarget point_385_contact:=[[280,137,134.5],[0,0,1,0],[0, 0, 0, 0],[9E+09,9E+09,9E+09,9E+09,9E+09,9E+09]];
    CONST robtarget point_385_clearance:=[[280,137,149.5],[0,0,1,0],[0, 0, 0, 0],[9E+09,9E+09,9E+09,9E+09,9E+09,9E+09]];
    CONST robtarget point_386_clearance:=[[425,153,149.5],[0,0,1,0],[0, 0, 0, 0],[9E+09,9E+09,9E+09,9E+09,9E+09,9E+09]];
    CONST robtarget point_386_contact:=[[425,153,134.5],[0,0,1,0],[0, 0, 0, 0],[9E+09,9E+09,9E+09,9E+09,9E+09,9E+09]];
    CONST robtarget point_387_contact:=[[424,130,134.5],[0,0,1,0],[0, 0, 0, 0],[9E+09,9E+09,9E+09,9E+09,9E+09,9E+09]];
    CONST robtarget point_387_clearance:=[[424,130,149.5],[0,0,1,0],[0, 0, 0, 0],[9E+09,9E+09,9E+09,9E+09,9E+09,9E+09]];
    CONST robtarget point_388_clearance:=[[322,136,149.5],[0,0,1,0],[0, 0, 0, 0],[9E+09,9E+09,9E+09,9E+09,9E+09,9E+09]];
    CONST robtarget point_388_contact:=[[322,136,134.5],[0,0,1,0],[0, 0, 0, 0],[9E+09,9E+09,9E+09,9E+09,9E+09,9E+09]];
    CONST robtarget point_389_contact:=[[311,134,134.5],[0,0,1,0],[0, 0, 0, 0],[9E+09,9E+09,9E+09,9E+09,9E+09,9E+09]];
    CONST robtarget point_389_clearance:=[[311,134,149.5],[0,0,1,0],[0, 0, 0, 0],[9E+09,9E+09,9E+09,9E+09,9E+09,9E+09]];
    CONST robtarget point_390_clearance:=[[377,136,149.5],[0,0,1,0],[0, 0, 0, 0],[9E+09,9E+09,9E+09,9E+09,9E+09,9E+09]];
    CONST robtarget point_390_contact:=[[377,136,134.5],[0,0,1,0],[0, 0, 0, 0],[9E+09,9E+09,9E+09,9E+09,9E+09,9E+09]];
    CONST robtarget point_391_contact:=[[386,133,134.5],[0,0,1,0],[0, 0, 0, 0],[9E+09,9E+09,9E+09,9E+09,9E+09,9E+09]];
    CONST robtarget point_391_clearance:=[[386,133,149.5],[0,0,1,0],[0, 0, 0, 0],[9E+09,9E+09,9E+09,9E+09,9E+09,9E+09]];
    CONST robtarget point_392_clearance:=[[321,136,149.5],[0,0,1,0],[0, 0, 0, 0],[9E+09,9E+09,9E+09,9E+09,9E+09,9E+09]];
    CONST robtarget point_392_contact:=[[321,136,134.5],[0,0,1,0],[0, 0, 0, 0],[9E+09,9E+09,9E+09,9E+09,9E+09,9E+09]];
    CONST robtarget point_393_contact:=[[334,135,134.5],[0,0,1,0],[0, 0, 0, 0],[9E+09,9E+09,9E+09,9E+09,9E+09,9E+09]];
    CONST robtarget point_393_clearance:=[[334,135,149.5],[0,0,1,0],[0, 0, 0, 0],[9E+09,9E+09,9E+09,9E+09,9E+09,9E+09]];
    CONST robtarget point_394_clearance:=[[429,132,149.5],[0,0,1,0],[0, 0, 0, 0],[9E+09,9E+09,9E+09,9E+09,9E+09,9E+09]];
    CONST robtarget point_394_contact:=[[429,132,134.5],[0,0,1,0],[0, 0, 0, 0],[9E+09,9E+09,9E+09,9E+09,9E+09,9E+09]];
    CONST robtarget point_395_contact:=[[431,182,134.5],[0,0,1,0],[0, 0, 0, 0],[9E+09,9E+09,9E+09,9E+09,9E+09,9E+09]];
    CONST robtarget point_395_clearance:=[[431,182,149.5],[0,0,1,0],[0, 0, 0, 0],[9E+09,9E+09,9E+09,9E+09,9E+09,9E+09]];
    CONST robtarget point_396_clearance:=[[256,137,149.5],[0,0,1,0],[0, 0, 0, 0],[9E+09,9E+09,9E+09,9E+09,9E+09,9E+09]];
    CONST robtarget point_396_contact:=[[256,137,134.5],[0,0,1,0],[0, 0, 0, 0],[9E+09,9E+09,9E+09,9E+09,9E+09,9E+09]];
    CONST robtarget point_397_contact:=[[265,135,134.5],[0,0,1,0],[0, 0, 0, 0],[9E+09,9E+09,9E+09,9E+09,9E+09,9E+09]];
    CONST robtarget point_397_clearance:=[[265,135,149.5],[0,0,1,0],[0, 0, 0, 0],[9E+09,9E+09,9E+09,9E+09,9E+09,9E+09]];
    CONST robtarget point_398_clearance:=[[343,150,149.5],[0,0,1,0],[0, 0, 0, 0],[9E+09,9E+09,9E+09,9E+09,9E+09,9E+09]];
    CONST robtarget point_398_contact:=[[343,150,134.5],[0,0,1,0],[0, 0, 0, 0],[9E+09,9E+09,9E+09,9E+09,9E+09,9E+09]];
    CONST robtarget point_399_contact:=[[339,133,134.5],[0,0,1,0],[0, 0, 0, 0],[9E+09,9E+09,9E+09,9E+09,9E+09,9E+09]];
    CONST robtarget point_399_clearance:=[[339,133,149.5],[0,0,1,0],[0, 0, 0, 0],[9E+09,9E+09,9E+09,9E+09,9E+09,9E+09]];
    CONST robtarget point_400_clearance:=[[179,140,149.5],[0,0,1,0],[0, 0, 0, 0],[9E+09,9E+09,9E+09,9E+09,9E+09,9E+09]];
    CONST robtarget point_400_contact:=[[179,140,134.5],[0,0,1,0],[0, 0, 0, 0],[9E+09,9E+09,9E+09,9E+09,9E+09,9E+09]];
    CONST robtarget point_401_contact:=[[168,135,134.5],[0,0,1,0],[0, 0, 0, 0],[9E+09,9E+09,9E+09,9E+09,9E+09,9E+09]];
    CONST robtarget point_401_clearance:=[[168,135,149.5],[0,0,1,0],[0, 0, 0, 0],[9E+09,9E+09,9E+09,9E+09,9E+09,9E+09]];
    CONST robtarget point_402_clearance:=[[192,156,149.5],[0,0,1,0],[0, 0, 0, 0],[9E+09,9E+09,9E+09,9E+09,9E+09,9E+09]];
    CONST robtarget point_402_contact:=[[192,156,134.5],[0,0,1,0],[0, 0, 0, 0],[9E+09,9E+09,9E+09,9E+09,9E+09,9E+09]];
    CONST robtarget point_403_contact:=[[195,135,134.5],[0,0,1,0],[0, 0, 0, 0],[9E+09,9E+09,9E+09,9E+09,9E+09,9E+09]];
    CONST robtarget point_403_clearance:=[[195,135,149.5],[0,0,1,0],[0, 0, 0, 0],[9E+09,9E+09,9E+09,9E+09,9E+09,9E+09]];
    CONST robtarget point_404_clearance:=[[198,145,149.5],[0,0,1,0],[0, 0, 0, 0],[9E+09,9E+09,9E+09,9E+09,9E+09,9E+09]];
    CONST robtarget point_404_contact:=[[198,145,134.5],[0,0,1,0],[0, 0, 0, 0],[9E+09,9E+09,9E+09,9E+09,9E+09,9E+09]];
    CONST robtarget point_405_contact:=[[200,135,134.5],[0,0,1,0],[0, 0, 0, 0],[9E+09,9E+09,9E+09,9E+09,9E+09,9E+09]];
    CONST robtarget point_405_clearance:=[[200,135,149.5],[0,0,1,0],[0, 0, 0, 0],[9E+09,9E+09,9E+09,9E+09,9E+09,9E+09]];
    CONST robtarget point_406_clearance:=[[202,136,149.5],[0,0,1,0],[0, 0, 0, 0],[9E+09,9E+09,9E+09,9E+09,9E+09,9E+09]];
    CONST robtarget point_406_contact:=[[202,136,134.5],[0,0,1,0],[0, 0, 0, 0],[9E+09,9E+09,9E+09,9E+09,9E+09,9E+09]];
    CONST robtarget point_407_contact:=[[203,163,134.5],[0,0,1,0],[0, 0, 0, 0],[9E+09,9E+09,9E+09,9E+09,9E+09,9E+09]];
    CONST robtarget point_407_clearance:=[[203,163,149.5],[0,0,1,0],[0, 0, 0, 0],[9E+09,9E+09,9E+09,9E+09,9E+09,9E+09]];
    CONST robtarget point_408_clearance:=[[231,138,149.5],[0,0,1,0],[0, 0, 0, 0],[9E+09,9E+09,9E+09,9E+09,9E+09,9E+09]];
    CONST robtarget point_408_contact:=[[231,138,134.5],[0,0,1,0],[0, 0, 0, 0],[9E+09,9E+09,9E+09,9E+09,9E+09,9E+09]];
    CONST robtarget point_409_contact:=[[237,140,134.5],[0,0,1,0],[0, 0, 0, 0],[9E+09,9E+09,9E+09,9E+09,9E+09,9E+09]];
    CONST robtarget point_409_clearance:=[[237,140,149.5],[0,0,1,0],[0, 0, 0, 0],[9E+09,9E+09,9E+09,9E+09,9E+09,9E+09]];
    CONST robtarget point_410_clearance:=[[311,138,149.5],[0,0,1,0],[0, 0, 0, 0],[9E+09,9E+09,9E+09,9E+09,9E+09,9E+09]];
    CONST robtarget point_410_contact:=[[311,138,134.5],[0,0,1,0],[0, 0, 0, 0],[9E+09,9E+09,9E+09,9E+09,9E+09,9E+09]];
    CONST robtarget point_411_contact:=[[302,137,134.5],[0,0,1,0],[0, 0, 0, 0],[9E+09,9E+09,9E+09,9E+09,9E+09,9E+09]];
    CONST robtarget point_411_clearance:=[[302,137,149.5],[0,0,1,0],[0, 0, 0, 0],[9E+09,9E+09,9E+09,9E+09,9E+09,9E+09]];
    CONST robtarget point_412_clearance:=[[143,158,149.5],[0,0,1,0],[0, 0, 0, 0],[9E+09,9E+09,9E+09,9E+09,9E+09,9E+09]];
    CONST robtarget point_412_contact:=[[143,158,134.5],[0,0,1,0],[0, 0, 0, 0],[9E+09,9E+09,9E+09,9E+09,9E+09,9E+09]];
    CONST robtarget point_413_contact:=[[142,137,134.5],[0,0,1,0],[0, 0, 0, 0],[9E+09,9E+09,9E+09,9E+09,9E+09,9E+09]];
    CONST robtarget point_413_clearance:=[[142,137,149.5],[0,0,1,0],[0, 0, 0, 0],[9E+09,9E+09,9E+09,9E+09,9E+09,9E+09]];
    CONST robtarget point_414_clearance:=[[206,145,149.5],[0,0,1,0],[0, 0, 0, 0],[9E+09,9E+09,9E+09,9E+09,9E+09,9E+09]];
